gfCNCPoint1[14456] = {X 450.4384, Y 41.0287, Z -1.3333, A 0.000, B 0.000, C 0.000 }
gfCNCPoint1[14457] = {X 450.4384, Y 34.2338, Z -1.3333, A 0.000, B 0.000, C 0.000 }
gfCNCPoint1[14458] = {X 447.3268, Y 34.2338, Z -1.3333, A 0.000, B 0.000, C 0.000 }
gfCNCPoint1[14459] = {X 442.9270, Y 42.8001, Z -1.3333, A 0.000, B 0.000, C 0.000 }
gfCNCPoint1[14460] = {X 442.9680, Y 42.9095, Z -1.3333, A 0.000, B 0.000, C 0.000 }
gfCNCPoint1[14461] = {X 443.1240, Y 43.5326, Z -1.3333, A 0.000, B 0.000, C 0.000 }
gfCNCPoint1[14462] = {X 443.1803, Y 44.1725, Z -1.3333, A 0.000, B 0.000, C 0.000 }
gfCNCPoint1[14463] = {X 443.1805, Y 45.0000, Z -1.3333, A 0.000, B 0.000, C 0.000 }
gfCNCPoint1[14464] = {X 443.0782, Y 45.9079, Z -1.3333, A 0.000, B 0.000, C 0.000 }
gfCNCPoint1[14465] = {X 442.7764, Y 46.7702, Z -1.3333, A 0.000, B 0.000, C 0.000 }
gfCNCPoint1[14466] = {X 442.2903, Y 47.5438, Z -1.3333, A 0.000, B 0.000, C 0.000 }
gfCNCPoint1[14467] = {X 441.6443, Y 48.1899, Z -1.3333, A 0.000, B 0.000, C 0.000 }
gfCNCPoint1[14468] = {X 440.8707, Y 48.6760, Z -1.3333, A 0.000, B 0.000, C 0.000 }
gfCNCPoint1[14469] = {X 440.0084, Y 48.9777, Z -1.3333, A 0.000, B 0.000, C 0.000 }
gfCNCPoint1[14470] = {X 439.1005, Y 49.0800, Z -1.3333, A 0.000, B 0.000, C 0.000 }
gfCNCPoint1[14471] = {X 432.5144, Y 49.0800, Z -1.3333, A 0.000, B 0.000, C 0.000 }
gfCNCPoint1[14472] = {X 431.6065, Y 48.9777, Z -1.3333, A 0.000, B 0.000, C 0.000 }
gfCNCPoint1[14473] = {X 430.7442, Y 48.6760, Z -1.3333, A 0.000, B 0.000, C 0.000 }
gfCNCPoint1[14474] = {X 429.9706, Y 48.1899, Z -1.3333, A 0.000, B 0.000, C 0.000 }
gfCNCPoint1[14475] = {X 429.3245, Y 47.5438, Z -1.3333, A 0.000, B 0.000, C 0.000 }
gfCNCPoint1[14476] = {X 428.8385, Y 46.7702, Z -1.3333, A 0.000, B 0.000, C 0.000 }
gfCNCPoint1[14477] = {X 428.5367, Y 45.9079, Z -1.3333, A 0.000, B 0.000, C 0.000 }
gfCNCPoint1[14478] = {X 428.4344, Y 45.0000, Z -1.3333, A 0.000, B 0.000, C 0.000 }
gfCNCPoint1[14479] = {X 428.4348, Y 44.1527, Z -1.3333, A 0.000, B 0.000, C 0.000 }
gfCNCPoint1[14480] = {X 428.5303, Y 43.3294, Z -1.3333, A 0.000, B 0.000, C 0.000 }
gfCNCPoint1[14481] = {X 428.7902, Y 42.5424, Z -1.3333, A 0.000, B 0.000, C 0.000 }
gfCNCPoint1[14482] = {X 429.2038, Y 41.8242, Z -1.3333, A 0.000, B 0.000, C 0.000 }
gfCNCPoint1[14483] = {X 429.7540, Y 41.2044, Z -1.3333, A 0.000, B 0.000, C 0.000 }
gfCNCPoint1[14484] = {X 430.4181, Y 40.7085, Z -1.3333, A 0.000, B 0.000, C 0.000 }
gfCNCPoint1[14485] = {X 431.1687, Y 40.3571, Z -1.3333, A 0.000, B 0.000, C 0.000 }
gfCNCPoint1[14486] = {X 435.3054, Y 32.2601, Z -1.3333, A 0.000, B 0.000, C 0.000 }
gfCNCPoint1[14487] = {X 434.1145, Y 31.4915, Z -1.3333, A 0.000, B 0.000, C 0.000 }
gfCNCPoint1[14488] = {X 433.0315, Y 30.5771, Z -1.3333, A 0.000, B 0.000, C 0.000 }
gfCNCPoint1[14489] = {X 432.0741, Y 29.5320, Z -1.3333, A 0.000, B 0.000, C 0.000 }
gfCNCPoint1[14490] = {X 431.2580, Y 28.3732, Z -1.3333, A 0.000, B 0.000, C 0.000 }
gfCNCPoint1[14491] = {X 430.5964, Y 27.1197, Z -1.3333, A 0.000, B 0.000, C 0.000 }
gfCNCPoint1[14492] = {X 430.1003, Y 25.7920, Z -1.3333, A 0.000, B 0.000, C 0.000 }
gfCNCPoint1[14493] = {X 429.6876, Y 24.0071, Z -1.3333, A 0.000, B 0.000, C 0.000 }
gfCNCPoint1[14494] = {X 429.4774, Y 22.1872, Z -1.3333, A 0.000, B 0.000, C 0.000 }
gfCNCPoint1[14495] = {X 429.4722, Y 20.3552, Z -1.3333, A 0.000, B 0.000, C 0.000 }
gfCNCPoint1[14496] = {X 429.6722, Y 18.5341, Z -1.3333, A 0.000, B 0.000, C 0.000 }
gfCNCPoint1[14497] = {X 430.0749, Y 16.7469, Z -1.3333, A 0.000, B 0.000, C 0.000 }
gfCNCPoint1[14498] = {X 430.5856, Y 15.3070, Z -1.3333, A 0.000, B 0.000, C 0.000 }
gfCNCPoint1[14499] = {X 431.2819, Y 13.9471, Z -1.3333, A 0.000, B 0.000, C 0.000 }
gfCNCPoint1[14500] = {X 432.1516, Y 12.6910, Z -1.3333, A 0.000, B 0.000, C 0.000 }
gfCNCPoint1[14501] = {X 433.1794, Y 11.5607, Z -1.3333, A 0.000, B 0.000, C 0.000 }
gfCNCPoint1[14502] = {X 434.3473, Y 10.5759, Z -1.3333, A 0.000, B 0.000, C 0.000 }
gfCNCPoint1[14503] = {X 435.6351, Y 9.7538, Z -1.3333, A 0.000, B 0.000, C 0.000 }
gfCNCPoint1[14504] = {X 437.0200, Y 9.1088, Z -1.3333, A 0.000, B 0.000, C 0.000 }
gfCNCPoint1[14505] = {X 438.4780, Y 8.6523, Z -1.3333, A 0.000, B 0.000, C 0.000 }
gfCNCPoint1[14506] = {X 440.0844, Y 8.3468, Z -1.3333, A 0.000, B 0.000, C 0.000 }
gfCNCPoint1[14507] = {X 441.7098, Y 8.1677, Z -1.3333, A 0.000, B 0.000, C 0.000 }
gfCNCPoint1[14508] = {X 443.3442, Y 8.1160, Z -1.3333, A 0.000, B 0.000, C 0.000 }
gfCNCPoint1[14509] = {X 444.0364, Y 8.1119, Z -1.3333, A 0.000, B 0.000, C 0.000 }
gfCNCPoint1[14510] = {X 459.4465, Y 8.1119, Z -1.3333, A 0.000, B 0.000, C 0.000 }
gfCNCPoint1[14511] = {X 460.3525, Y 8.2140, Z -1.3333, A 0.000, B 0.000, C 0.000 }
gfCNCPoint1[14512] = {X 461.2130, Y 8.5151, Z -1.3333, A 0.000, B 0.000, C 0.000 }
gfCNCPoint1[14513] = {X 461.9850, Y 9.0002, Z -1.3333, A 0.000, B 0.000, C 0.000 }
gfCNCPoint1[14514] = {X 462.6297, Y 9.6448, Z -1.3333, A 0.000, B 0.000, C 0.000 }
gfCNCPoint1[14515] = {X 463.1147, Y 10.4168, Z -1.3333, A 0.000, B 0.000, C 0.000 }
gfCNCPoint1[14516] = {X 463.4159, Y 11.2774, Z -1.3333, A 0.000, B 0.000, C 0.000 }
gfCNCPoint1[14517] = {X 463.5179, Y 12.1834, Z -1.3333, A 0.000, B 0.000, C 0.000 }
gfCNCPoint1[14518] = {X 463.5179, Y 12.9781, Z -1.3333, A 0.000, B 0.000, C 0.000 }
gfCNCPoint1[14519] = {X 463.4240, Y 13.8483, Z -1.3333, A 0.000, B 0.000, C 0.000 }
gfCNCPoint1[14520] = {X 463.1467, Y 14.6785, Z -1.3333, A 0.000, B 0.000, C 0.000 }
gfCNCPoint1[14521] = {X 462.6987, Y 15.4304, Z -1.3333, A 0.000, B 0.000, C 0.000 }
gfCNCPoint1[14522] = {X 462.1006, Y 16.0694, Z -1.3333, A 0.000, B 0.000, C 0.000 }
gfCNCPoint1[14523] = {X 462.0432, Y 16.1179, Z -1.3333, A 0.000, B 0.000, C 0.000 }
gfCNCPoint1[14524] = {X 461.9850, Y 16.1653, Z -1.3333, A 0.000, B 0.000, C 0.000 }
gfCNCPoint1[14525] = {X 461.9894, Y 16.2000, Z -1.3333, A 0.000, B 0.000, C 0.000 }
gfCNCPoint1[14526] = {X 461.9896, Y 28.5936, Z -1.3333, A 0.000, B 0.000, C 0.000 }
gfCNCPoint1[14527] = {X 465.9896, Y 28.5935, Z -1.3333, A 0.000, B 0.000, C 0.000 }
gfCNCPoint1[14528] = {X 461.9096, Y 28.5936, Z -1.3333, A 0.000, B 0.000, C 0.000 }
gfCNCPoint1[14529] = {X 461.9098, Y 41.0659, Z -1.3333, A 0.000, B 0.000, C 0.000 }
gfCNCPoint1[14530] = {X 462.0488, Y 41.1783, Z -1.3333, A 0.000, B 0.000, C 0.000 }
gfCNCPoint1[14531] = {X 462.6350, Y 41.8049, Z -1.3333, A 0.000, B 0.000, C 0.000 }
gfCNCPoint1[14532] = {X 463.0741, Y 42.5420, Z -1.3333, A 0.000, B 0.000, C 0.000 }
gfCNCPoint1[14533] = {X 463.3459, Y 43.3558, Z -1.3333, A 0.000, B 0.000, C 0.000 }
gfCNCPoint1[14534] = {X 463.4379, Y 44.2089, Z -1.3333, A 0.000, B 0.000, C 0.000 }
gfCNCPoint1[14535] = {X 463.4379, Y 45.0000, Z -1.3333, A 0.000, B 0.000, C 0.000 }
gfCNCPoint1[14536] = {X 463.3377, Y 45.8901, Z -1.3333, A 0.000, B 0.000, C 0.000 }
gfCNCPoint1[14537] = {X 463.0418, Y 46.7355, Z -1.3333, A 0.000, B 0.000, C 0.000 }
gfCNCPoint1[14538] = {X 462.5653, Y 47.4940, Z -1.3333, A 0.000, B 0.000, C 0.000 }
gfCNCPoint1[14539] = {X 461.9319, Y 48.1273, Z -1.3333, A 0.000, B 0.000, C 0.000 }
gfCNCPoint1[14540] = {X 461.1735, Y 48.6039, Z -1.3333, A 0.000, B 0.000, C 0.000 }
gfCNCPoint1[14541] = {X 460.3280, Y 48.8997, Z -1.3333, A 0.000, B 0.000, C 0.000 }
gfCNCPoint1[14542] = {X 459.4379, Y 49.0000, Z -1.3333, A 0.000, B 0.000, C 0.000 }
gfCNCPoint1[14543] = {X 452.9945, Y 49.0000, Z -1.3333, A 0.000, B 0.000, C 0.000 }
gfCNCPoint1[14544] = {X 452.1044, Y 48.8997, Z -1.3333, A 0.000, B 0.000, C 0.000 }
gfCNCPoint1[14545] = {X 451.2589, Y 48.6039, Z -1.3333, A 0.000, B 0.000, C 0.000 }
gfCNCPoint1[14546] = {X 450.5005, Y 48.1273, Z -1.3333, A 0.000, B 0.000, C 0.000 }
gfCNCPoint1[14547] = {X 449.8671, Y 47.4939, Z -1.3333, A 0.000, B 0.000, C 0.000 }
gfCNCPoint1[14548] = {X 449.3906, Y 46.7355, Z -1.3333, A 0.000, B 0.000, C 0.000 }
gfCNCPoint1[14549] = {X 449.0948, Y 45.8900, Z -1.3333, A 0.000, B 0.000, C 0.000 }
gfCNCPoint1[14550] = {X 448.9945, Y 44.9999, Z -1.3333, A 0.000, B 0.000, C 0.000 }
gfCNCPoint1[14551] = {X 448.9949, Y 44.1538, Z -1.3333, A 0.000, B 0.000, C 0.000 }
gfCNCPoint1[14552] = {X 449.1055, Y 43.2730, Z -1.3333, A 0.000, B 0.000, C 0.000 }
gfCNCPoint1[14553] = {X 449.4077, Y 42.4382, Z -1.3333, A 0.000, B 0.000, C 0.000 }
gfCNCPoint1[14554] = {X 449.8865, Y 41.6907, Z -1.3333, A 0.000, B 0.000, C 0.000 }
gfCNCPoint1[14555] = {X 450.5184, Y 41.0672, Z -1.3333, A 0.000, B 0.000, C 0.000 }
gfCNCPoint1[14556] = {X 450.5184, Y 34.1538, Z -1.3333, A 0.000, B 0.000, C 0.000 }
gfCNCPoint1[14557] = {X 447.5222, Y 34.1538, Z -1.3333, A 0.000, B 0.000, C 0.000 }
gfCNCPoint1[14558] = {X 447.2789, Y 34.1521, Z -1.3333, A 0.000, B 0.000, C 0.000 }
gfCNCPoint1[14559] = {X 442.8397, Y 42.7950, Z -1.3333, A 0.000, B 0.000, C 0.000 }
gfCNCPoint1[14560] = {X 442.8963, Y 42.9473, Z -1.3333, A 0.000, B 0.000, C 0.000 }
gfCNCPoint1[14561] = {X 443.0491, Y 43.5699, Z -1.3333, A 0.000, B 0.000, C 0.000 }
gfCNCPoint1[14562] = {X 443.1005, Y 44.2089, Z -1.3333, A 0.000, B 0.000, C 0.000 }
gfCNCPoint1[14563] = {X 443.1005, Y 45.0000, Z -1.3333, A 0.000, B 0.000, C 0.000 }
gfCNCPoint1[14564] = {X 443.0002, Y 45.8901, Z -1.3333, A 0.000, B 0.000, C 0.000 }
gfCNCPoint1[14565] = {X 442.7043, Y 46.7355, Z -1.3333, A 0.000, B 0.000, C 0.000 }
gfCNCPoint1[14566] = {X 442.2278, Y 47.4940, Z -1.3333, A 0.000, B 0.000, C 0.000 }
gfCNCPoint1[14567] = {X 441.5944, Y 48.1273, Z -1.3333, A 0.000, B 0.000, C 0.000 }
gfCNCPoint1[14568] = {X 440.8360, Y 48.6039, Z -1.3333, A 0.000, B 0.000, C 0.000 }
gfCNCPoint1[14569] = {X 439.9906, Y 48.8997, Z -1.3333, A 0.000, B 0.000, C 0.000 }
gfCNCPoint1[14570] = {X 439.1005, Y 49.0000, Z -1.3333, A 0.000, B 0.000, C 0.000 }
gfCNCPoint1[14571] = {X 432.5144, Y 49.0000, Z -1.3333, A 0.000, B 0.000, C 0.000 }
gfCNCPoint1[14572] = {X 431.6243, Y 48.8997, Z -1.3333, A 0.000, B 0.000, C 0.000 }
gfCNCPoint1[14573] = {X 430.7789, Y 48.6039, Z -1.3333, A 0.000, B 0.000, C 0.000 }
gfCNCPoint1[14574] = {X 430.0204, Y 48.1273, Z -1.3333, A 0.000, B 0.000, C 0.000 }
gfCNCPoint1[14575] = {X 429.3871, Y 47.4940, Z -1.3333, A 0.000, B 0.000, C 0.000 }
gfCNCPoint1[14576] = {X 428.9105, Y 46.7355, Z -1.3333, A 0.000, B 0.000, C 0.000 }
gfCNCPoint1[14577] = {X 428.6147, Y 45.8901, Z -1.3333, A 0.000, B 0.000, C 0.000 }
gfCNCPoint1[14578] = {X 428.5144, Y 45.0000, Z -1.3333, A 0.000, B 0.000, C 0.000 }
gfCNCPoint1[14579] = {X 428.5148, Y 44.1538, Z -1.3333, A 0.000, B 0.000, C 0.000 }
gfCNCPoint1[14580] = {X 428.6096, Y 43.3414, Z -1.3333, A 0.000, B 0.000, C 0.000 }
gfCNCPoint1[14581] = {X 428.8676, Y 42.5654, Z -1.3333, A 0.000, B 0.000, C 0.000 }
gfCNCPoint1[14582] = {X 429.2781, Y 41.8580, Z -1.3333, A 0.000, B 0.000, C 0.000 }
gfCNCPoint1[14583] = {X 429.8239, Y 41.2489, Z -1.3333, A 0.000, B 0.000, C 0.000 }
gfCNCPoint1[14584] = {X 430.4821, Y 40.7635, Z -1.3333, A 0.000, B 0.000, C 0.000 }
gfCNCPoint1[14585] = {X 431.2253, Y 40.4222, Z -1.3333, A 0.000, B 0.000, C 0.000 }
gfCNCPoint1[14586] = {X 435.4118, Y 32.2276, Z -1.3333, A 0.000, B 0.000, C 0.000 }
gfCNCPoint1[14587] = {X 434.2139, Y 31.4652, Z -1.3333, A 0.000, B 0.000, C 0.000 }
gfCNCPoint1[14588] = {X 433.1241, Y 30.5549, Z -1.3333, A 0.000, B 0.000, C 0.000 }
gfCNCPoint1[14589] = {X 432.1607, Y 29.5118, Z -1.3333, A 0.000, B 0.000, C 0.000 }
gfCNCPoint1[14590] = {X 431.3397, Y 28.3533, Z -1.3333, A 0.000, B 0.000, C 0.000 }
gfCNCPoint1[14591] = {X 430.6747, Y 27.0987, Z -1.3333, A 0.000, B 0.000, C 0.000 }
gfCNCPoint1[14592] = {X 430.1769, Y 25.7689, Z -1.3333, A 0.000, B 0.000, C 0.000 }
gfCNCPoint1[14593] = {X 429.7663, Y 23.9928, Z -1.3333, A 0.000, B 0.000, C 0.000 }
gfCNCPoint1[14594] = {X 429.5572, Y 22.1819, Z -1.3333, A 0.000, B 0.000, C 0.000 }
gfCNCPoint1[14595] = {X 429.5521, Y 20.3591, Z -1.3333, A 0.000, B 0.000, C 0.000 }
gfCNCPoint1[14596] = {X 429.7512, Y 18.5471, Z -1.3333, A 0.000, B 0.000, C 0.000 }
gfCNCPoint1[14597] = {X 430.1519, Y 16.7687, Z -1.3333, A 0.000, B 0.000, C 0.000 }
gfCNCPoint1[14598] = {X 430.6590, Y 15.3388, Z -1.3333, A 0.000, B 0.000, C 0.000 }
gfCNCPoint1[14599] = {X 431.3505, Y 13.9883, Z -1.3333, A 0.000, B 0.000, C 0.000 }
gfCNCPoint1[14600] = {X 432.2141, Y 12.7409, Z -1.3333, A 0.000, B 0.000, C 0.000 }
gfCNCPoint1[14601] = {X 433.2348, Y 11.6184, Z -1.3333, A 0.000, B 0.000, C 0.000 }
gfCNCPoint1[14602] = {X 434.3947, Y 10.6403, Z -1.3333, A 0.000, B 0.000, C 0.000 }
gfCNCPoint1[14603] = {X 435.6735, Y 9.8239, Z -1.3333, A 0.000, B 0.000, C 0.000 }
gfCNCPoint1[14604] = {X 437.0489, Y 9.1834, Z -1.3333, A 0.000, B 0.000, C 0.000 }
gfCNCPoint1[14605] = {X 438.4968, Y 8.7301, Z -1.3333, A 0.000, B 0.000, C 0.000 }
gfCNCPoint1[14606] = {X 440.0970, Y 8.4258, Z -1.3333, A 0.000, B 0.000, C 0.000 }
gfCNCPoint1[14607] = {X 441.7161, Y 8.2474, Z -1.3333, A 0.000, B 0.000, C 0.000 }
gfCNCPoint1[14608] = {X 443.3442, Y 8.1960, Z -1.3333, A 0.000, B 0.000, C 0.000 }
gfCNCPoint1[14609] = {X 444.0367, Y 8.1919, Z -1.3333, A 0.000, B 0.000, C 0.000 }
gfCNCPoint1[14610] = {X 459.4465, Y 8.1919, Z -1.3333, A 0.000, B 0.000, C 0.000 }
gfCNCPoint1[14611] = {X 460.3347, Y 8.2920, Z -1.3333, A 0.000, B 0.000, C 0.000 }
gfCNCPoint1[14612] = {X 461.1783, Y 8.5872, Z -1.3333, A 0.000, B 0.000, C 0.000 }
gfCNCPoint1[14613] = {X 461.9351, Y 9.0627, Z -1.3333, A 0.000, B 0.000, C 0.000 }
gfCNCPoint1[14614] = {X 462.5671, Y 9.6947, Z -1.3333, A 0.000, B 0.000, C 0.000 }
gfCNCPoint1[14615] = {X 463.0427, Y 10.4515, Z -1.3333, A 0.000, B 0.000, C 0.000 }
gfCNCPoint1[14616] = {X 463.3379, Y 11.2952, Z -1.3333, A 0.000, B 0.000, C 0.000 }
gfCNCPoint1[14617] = {X 463.4379, Y 12.1834, Z -1.3333, A 0.000, B 0.000, C 0.000 }
gfCNCPoint1[14618] = {X 463.4378, Y 13.0163, Z -1.3333, A 0.000, B 0.000, C 0.000 }
gfCNCPoint1[14619] = {X 463.3397, Y 13.8592, Z -1.3333, A 0.000, B 0.000, C 0.000 }
gfCNCPoint1[14620] = {X 463.0660, Y 14.6625, Z -1.3333, A 0.000, B 0.000, C 0.000 }
gfCNCPoint1[14621] = {X 462.6290, Y 15.3899, Z -1.3333, A 0.000, B 0.000, C 0.000 }
gfCNCPoint1[14622] = {X 462.0484, Y 16.0088, Z -1.3333, A 0.000, B 0.000, C 0.000 }
gfCNCPoint1[14623] = {X 461.9721, Y 16.0729, Z -1.3333, A 0.000, B 0.000, C 0.000 }
gfCNCPoint1[14624] = {X 461.8942, Y 16.1351, Z -1.3333, A 0.000, B 0.000, C 0.000 }
gfCNCPoint1[14625] = {X 461.9094, Y 16.1924, Z -1.3333, A 0.000, B 0.000, C 0.000 }
gfCNCPoint1[14626] = {X 461.9096, Y 28.5936, Z -1.3333, A 0.000, B 0.000, C 0.000 }
gfCNCPoint1[14627] = {X 465.9896, Y 28.5935, Z -1.3333, A 0.000, B 0.000, C 0.000 }
gfCNCPoint1[14628] = {X 465.9896, Y 28.5935, Z 1.6667, A 0.000, B 0.000, C 0.000 }
gfCNCPoint1[14629] = {X 465.9896, Y 28.5935, Z 11.0000, A 0.000, B 0.000, C 0.000 }
gfCNCPoint1[14630] = {X 492.3824, Y 3.7919, Z 11.0000, A 0.000, B 0.000, C 0.000 }
gfCNCPoint1[14631] = {X 492.3824, Y 3.7919, Z 1.6667, A 0.000, B 0.000, C 0.000 }
gfCNCPoint1[14632] = {X 492.3824, Y 3.7919, Z -1.3333, A 0.000, B 0.000, C 0.000 }
gfCNCPoint1[14633] = {X 492.3824, Y 7.8719, Z -1.3333, A 0.000, B 0.000, C 0.000 }
gfCNCPoint1[14634] = {X 502.2066, Y 7.8719, Z -1.3333, A 0.000, B 0.000, C 0.000 }
gfCNCPoint1[14635] = {X 502.7373, Y 7.8760, Z -1.3333, A 0.000, B 0.000, C 0.000 }
gfCNCPoint1[14636] = {X 503.6897, Y 7.9904, Z -1.3333, A 0.000, B 0.000, C 0.000 }
gfCNCPoint1[14637] = {X 504.5931, Y 8.3127, Z -1.3333, A 0.000, B 0.000, C 0.000 }
gfCNCPoint1[14638] = {X 505.4027, Y 8.8271, Z -1.3333, A 0.000, B 0.000, C 0.000 }
gfCNCPoint1[14639] = {X 506.0783, Y 9.5080, Z -1.3333, A 0.000, B 0.000, C 0.000 }
gfCNCPoint1[14640] = {X 506.5863, Y 10.3216, Z -1.3333, A 0.000, B 0.000, C 0.000 }
gfCNCPoint1[14641] = {X 506.9016, Y 11.2275, Z -1.3333, A 0.000, B 0.000, C 0.000 }
gfCNCPoint1[14642] = {X 507.0085, Y 12.1807, Z -1.3333, A 0.000, B 0.000, C 0.000 }
gfCNCPoint1[14643] = {X 507.0085, Y 12.9781, Z -1.3333, A 0.000, B 0.000, C 0.000 }
gfCNCPoint1[14644] = {X 506.9071, Y 13.9084, Z -1.3333, A 0.000, B 0.000, C 0.000 }
gfCNCPoint1[14645] = {X 506.6078, Y 14.7951, Z -1.3333, A 0.000, B 0.000, C 0.000 }
gfCNCPoint1[14646] = {X 506.1245, Y 15.5965, Z -1.3333, A 0.000, B 0.000, C 0.000 }
gfCNCPoint1[14647] = {X 505.4800, Y 16.2750, Z -1.3333, A 0.000, B 0.000, C 0.000 }
gfCNCPoint1[14648] = {X 505.4799, Y 40.9118, Z -1.3333, A 0.000, B 0.000, C 0.000 }
gfCNCPoint1[14649] = {X 506.1188, Y 41.5829, Z -1.3333, A 0.000, B 0.000, C 0.000 }
gfCNCPoint1[14650] = {X 506.5998, Y 42.3747, Z -1.3333, A 0.000, B 0.000, C 0.000 }
gfCNCPoint1[14651] = {X 506.9010, Y 43.2510, Z -1.3333, A 0.000, B 0.000, C 0.000 }
gfCNCPoint1[14652] = {X 507.0083, Y 44.1713, Z -1.3333, A 0.000, B 0.000, C 0.000 }
gfCNCPoint1[14653] = {X 507.0085, Y 45.0000, Z -1.3333, A 0.000, B 0.000, C 0.000 }
gfCNCPoint1[14654] = {X 506.9002, Y 45.9613, Z -1.3333, A 0.000, B 0.000, C 0.000 }
gfCNCPoint1[14655] = {X 506.5807, Y 46.8744, Z -1.3333, A 0.000, B 0.000, C 0.000 }
gfCNCPoint1[14656] = {X 506.0660, Y 47.6935, Z -1.3333, A 0.000, B 0.000, C 0.000 }
gfCNCPoint1[14657] = {X 505.3820, Y 48.3775, Z -1.3333, A 0.000, B 0.000, C 0.000 }
gfCNCPoint1[14658] = {X 504.5629, Y 48.8922, Z -1.3333, A 0.000, B 0.000, C 0.000 }
gfCNCPoint1[14659] = {X 503.6498, Y 49.2117, Z -1.3333, A 0.000, B 0.000, C 0.000 }
gfCNCPoint1[14660] = {X 502.6885, Y 49.3200, Z -1.3333, A 0.000, B 0.000, C 0.000 }
gfCNCPoint1[14661] = {X 496.2450, Y 49.3200, Z -1.3333, A 0.000, B 0.000, C 0.000 }
gfCNCPoint1[14662] = {X 495.2885, Y 49.2128, Z -1.3333, A 0.000, B 0.000, C 0.000 }
gfCNCPoint1[14663] = {X 494.3794, Y 48.8964, Z -1.3333, A 0.000, B 0.000, C 0.000 }
gfCNCPoint1[14664] = {X 493.5630, Y 48.3866, Z -1.3333, A 0.000, B 0.000, C 0.000 }
gfCNCPoint1[14665] = {X 492.8797, Y 47.7087, Z -1.3333, A 0.000, B 0.000, C 0.000 }
gfCNCPoint1[14666] = {X 492.3635, Y 46.8963, Z -1.3333, A 0.000, B 0.000, C 0.000 }
gfCNCPoint1[14667] = {X 492.0399, Y 45.9898, Z -1.3333, A 0.000, B 0.000, C 0.000 }
gfCNCPoint1[14668] = {X 491.9252, Y 45.0341, Z -1.3333, A 0.000, B 0.000, C 0.000 }
gfCNCPoint1[14669] = {X 491.9254, Y 44.1494, Z -1.3333, A 0.000, B 0.000, C 0.000 }
gfCNCPoint1[14670] = {X 492.0359, Y 43.2364, Z -1.3333, A 0.000, B 0.000, C 0.000 }
gfCNCPoint1[14671] = {X 492.3371, Y 42.3675, Z -1.3333, A 0.000, B 0.000, C 0.000 }
gfCNCPoint1[14672] = {X 492.8153, Y 41.5821, Z -1.3333, A 0.000, B 0.000, C 0.000 }
gfCNCPoint1[14673] = {X 493.4490, Y 40.9157, Z -1.3333, A 0.000, B 0.000, C 0.000 }
gfCNCPoint1[14674] = {X 493.4490, Y 34.4738, Z -1.3333, A 0.000, B 0.000, C 0.000 }
gfCNCPoint1[14675] = {X 490.7232, Y 34.4738, Z -1.3333, A 0.000, B 0.000, C 0.000 }
gfCNCPoint1[14676] = {X 486.4395, Y 42.8153, Z -1.3333, A 0.000, B 0.000, C 0.000 }
gfCNCPoint1[14677] = {X 486.4446, Y 42.8286, Z -1.3333, A 0.000, B 0.000, C 0.000 }
gfCNCPoint1[14678] = {X 486.6109, Y 43.4903, Z -1.3333, A 0.000, B 0.000, C 0.000 }
gfCNCPoint1[14679] = {X 486.6708, Y 44.1699, Z -1.3333, A 0.000, B 0.000, C 0.000 }
gfCNCPoint1[14680] = {X 486.6710, Y 45.0000, Z -1.3333, A 0.000, B 0.000, C 0.000 }
gfCNCPoint1[14681] = {X 486.5627, Y 45.9613, Z -1.3333, A 0.000, B 0.000, C 0.000 }
gfCNCPoint1[14682] = {X 486.2432, Y 46.8744, Z -1.3333, A 0.000, B 0.000, C 0.000 }
gfCNCPoint1[14683] = {X 485.7285, Y 47.6935, Z -1.3333, A 0.000, B 0.000, C 0.000 }
gfCNCPoint1[14684] = {X 485.0445, Y 48.3775, Z -1.3333, A 0.000, B 0.000, C 0.000 }
gfCNCPoint1[14685] = {X 484.2254, Y 48.8922, Z -1.3333, A 0.000, B 0.000, C 0.000 }
gfCNCPoint1[14686] = {X 483.3123, Y 49.2117, Z -1.3333, A 0.000, B 0.000, C 0.000 }
gfCNCPoint1[14687] = {X 482.3510, Y 49.3200, Z -1.3333, A 0.000, B 0.000, C 0.000 }
gfCNCPoint1[14688] = {X 475.7650, Y 49.3200, Z -1.3333, A 0.000, B 0.000, C 0.000 }
gfCNCPoint1[14689] = {X 474.8037, Y 49.2117, Z -1.3333, A 0.000, B 0.000, C 0.000 }
gfCNCPoint1[14690] = {X 473.8906, Y 48.8922, Z -1.3333, A 0.000, B 0.000, C 0.000 }
gfCNCPoint1[14691] = {X 473.0715, Y 48.3775, Z -1.3333, A 0.000, B 0.000, C 0.000 }
gfCNCPoint1[14692] = {X 472.3875, Y 47.6935, Z -1.3333, A 0.000, B 0.000, C 0.000 }
gfCNCPoint1[14693] = {X 471.8728, Y 46.8745, Z -1.3333, A 0.000, B 0.000, C 0.000 }
gfCNCPoint1[14694] = {X 471.5533, Y 45.9614, Z -1.3333, A 0.000, B 0.000, C 0.000 }
gfCNCPoint1[14695] = {X 471.4450, Y 45.0001, Z -1.3333, A 0.000, B 0.000, C 0.000 }
gfCNCPoint1[14696] = {X 471.4454, Y 44.1494, Z -1.3333, A 0.000, B 0.000, C 0.000 }
gfCNCPoint1[14697] = {X 471.5430, Y 43.2935, Z -1.3333, A 0.000, B 0.000, C 0.000 }
gfCNCPoint1[14698] = {X 471.8086, Y 42.4740, Z -1.3333, A 0.000, B 0.000, C 0.000 }
gfCNCPoint1[14699] = {X 472.2314, Y 41.7236, Z -1.3333, A 0.000, B 0.000, C 0.000 }
gfCNCPoint1[14700] = {X 472.7947, Y 41.0719, Z -1.3333, A 0.000, B 0.000, C 0.000 }
gfCNCPoint1[14701] = {X 473.4762, Y 40.5449, Z -1.3333, A 0.000, B 0.000, C 0.000 }
gfCNCPoint1[14702] = {X 474.2486, Y 40.1637, Z -1.3333, A 0.000, B 0.000, C 0.000 }
gfCNCPoint1[14703] = {X 478.2331, Y 32.3645, Z -1.3333, A 0.000, B 0.000, C 0.000 }
gfCNCPoint1[14704] = {X 476.9699, Y 31.4967, Z -1.3333, A 0.000, B 0.000, C 0.000 }
gfCNCPoint1[14705] = {X 475.8338, Y 30.4682, Z -1.3333, A 0.000, B 0.000, C 0.000 }
gfCNCPoint1[14706] = {X 474.8448, Y 29.2975, Z -1.3333, A 0.000, B 0.000, C 0.000 }
gfCNCPoint1[14707] = {X 474.0207, Y 28.0054, Z -1.3333, A 0.000, B 0.000, C 0.000 }
gfCNCPoint1[14708] = {X 473.3762, Y 26.6150, Z -1.3333, A 0.000, B 0.000, C 0.000 }
gfCNCPoint1[14709] = {X 472.9228, Y 25.1511, Z -1.3333, A 0.000, B 0.000, C 0.000 }
gfCNCPoint1[14710] = {X 472.6086, Y 23.4680, Z -1.3333, A 0.000, B 0.000, C 0.000 }
gfCNCPoint1[14711] = {X 472.4681, Y 21.7616, Z -1.3333, A 0.000, B 0.000, C 0.000 }
gfCNCPoint1[14712] = {X 472.5028, Y 20.0497, Z -1.3333, A 0.000, B 0.000, C 0.000 }
gfCNCPoint1[14713] = {X 472.7123, Y 18.3504, Z -1.3333, A 0.000, B 0.000, C 0.000 }
gfCNCPoint1[14714] = {X 473.0945, Y 16.6814, Z -1.3333, A 0.000, B 0.000, C 0.000 }
gfCNCPoint1[14715] = {X 473.6376, Y 15.1671, Z -1.3333, A 0.000, B 0.000, C 0.000 }
gfCNCPoint1[14716] = {X 474.3811, Y 13.7404, Z -1.3333, A 0.000, B 0.000, C 0.000 }
gfCNCPoint1[14717] = {X 475.3112, Y 12.4277, Z -1.3333, A 0.000, B 0.000, C 0.000 }
gfCNCPoint1[14718] = {X 476.4106, Y 11.2533, Z -1.3333, A 0.000, B 0.000, C 0.000 }
gfCNCPoint1[14719] = {X 477.6592, Y 10.2388, Z -1.3333, A 0.000, B 0.000, C 0.000 }
gfCNCPoint1[14720] = {X 479.0338, Y 9.4030, Z -1.3333, A 0.000, B 0.000, C 0.000 }
gfCNCPoint1[14721] = {X 480.5091, Y 8.7613, Z -1.3333, A 0.000, B 0.000, C 0.000 }
gfCNCPoint1[14722] = {X 482.0578, Y 8.3256, Z -1.3333, A 0.000, B 0.000, C 0.000 }
gfCNCPoint1[14723] = {X 484.1551, Y 7.9992, Z -1.3333, A 0.000, B 0.000, C 0.000 }
gfCNCPoint1[14724] = {X 486.2746, Y 7.8841, Z -1.3333, A 0.000, B 0.000, C 0.000 }
gfCNCPoint1[14725] = {X 486.9679, Y 7.8719, Z -1.3333, A 0.000, B 0.000, C 0.000 }
gfCNCPoint1[14726] = {X 492.3824, Y 7.8719, Z -1.3333, A 0.000, B 0.000, C 0.000 }
gfCNCPoint1[14727] = {X 492.3824, Y 3.8719, Z -1.3333, A 0.000, B 0.000, C 0.000 }
gfCNCPoint1[14728] = {X 492.3824, Y 7.9519, Z -1.3333, A 0.000, B 0.000, C 0.000 }
gfCNCPoint1[14729] = {X 502.2063, Y 7.9519, Z -1.3333, A 0.000, B 0.000, C 0.000 }
gfCNCPoint1[14730] = {X 502.7367, Y 7.9560, Z -1.3333, A 0.000, B 0.000, C 0.000 }
gfCNCPoint1[14731] = {X 503.6713, Y 8.0682, Z -1.3333, A 0.000, B 0.000, C 0.000 }
gfCNCPoint1[14732] = {X 504.5580, Y 8.3846, Z -1.3333, A 0.000, B 0.000, C 0.000 }
gfCNCPoint1[14733] = {X 505.3525, Y 8.8894, Z -1.3333, A 0.000, B 0.000, C 0.000 }
gfCNCPoint1[14734] = {X 506.0156, Y 9.5577, Z -1.3333, A 0.000, B 0.000, C 0.000 }
gfCNCPoint1[14735] = {X 506.5142, Y 10.3562, Z -1.3333, A 0.000, B 0.000, C 0.000 }
gfCNCPoint1[14736] = {X 506.8236, Y 11.2452, Z -1.3333, A 0.000, B 0.000, C 0.000 }
gfCNCPoint1[14737] = {X 506.9285, Y 12.1807, Z -1.3333, A 0.000, B 0.000, C 0.000 }
gfCNCPoint1[14738] = {X 506.9285, Y 12.9781, Z -1.3333, A 0.000, B 0.000, C 0.000 }
gfCNCPoint1[14739] = {X 506.8270, Y 13.9002, Z -1.3333, A 0.000, B 0.000, C 0.000 }
gfCNCPoint1[14740] = {X 506.5274, Y 14.7782, Z -1.3333, A 0.000, B 0.000, C 0.000 }
gfCNCPoint1[14741] = {X 506.0440, Y 15.5700, Z -1.3333, A 0.000, B 0.000, C 0.000 }
gfCNCPoint1[14742] = {X 505.4000, Y 16.2377, Z -1.3333, A 0.000, B 0.000, C 0.000 }
gfCNCPoint1[14743] = {X 505.3999, Y 40.9499, Z -1.3333, A 0.000, B 0.000, C 0.000 }
gfCNCPoint1[14744] = {X 505.4282, Y 40.9728, Z -1.3333, A 0.000, B 0.000, C 0.000 }
gfCNCPoint1[14745] = {X 506.0553, Y 41.6315, Z -1.3333, A 0.000, B 0.000, C 0.000 }
gfCNCPoint1[14746] = {X 506.5274, Y 42.4087, Z -1.3333, A 0.000, B 0.000, C 0.000 }
gfCNCPoint1[14747] = {X 506.8230, Y 43.2687, Z -1.3333, A 0.000, B 0.000, C 0.000 }
gfCNCPoint1[14748] = {X 506.9283, Y 44.1720, Z -1.3333, A 0.000, B 0.000, C 0.000 }
gfCNCPoint1[14749] = {X 506.9285, Y 45.0000, Z -1.3333, A 0.000, B 0.000, C 0.000 }
gfCNCPoint1[14750] = {X 506.8222, Y 45.9435, Z -1.3333, A 0.000, B 0.000, C 0.000 }
gfCNCPoint1[14751] = {X 506.5086, Y 46.8397, Z -1.3333, A 0.000, B 0.000, C 0.000 }
gfCNCPoint1[14752] = {X 506.0035, Y 47.6436, Z -1.3333, A 0.000, B 0.000, C 0.000 }
gfCNCPoint1[14753] = {X 505.3321, Y 48.3150, Z -1.3333, A 0.000, B 0.000, C 0.000 }
gfCNCPoint1[14754] = {X 504.5282, Y 48.8201, Z -1.3333, A 0.000, B 0.000, C 0.000 }
gfCNCPoint1[14755] = {X 503.6320, Y 49.1337, Z -1.3333, A 0.000, B 0.000, C 0.000 }
gfCNCPoint1[14756] = {X 502.6885, Y 49.2400, Z -1.3333, A 0.000, B 0.000, C 0.000 }
gfCNCPoint1[14757] = {X 496.2450, Y 49.2400, Z -1.3333, A 0.000, B 0.000, C 0.000 }
gfCNCPoint1[14758] = {X 495.3062, Y 49.1348, Z -1.3333, A 0.000, B 0.000, C 0.000 }
gfCNCPoint1[14759] = {X 494.4140, Y 48.8242, Z -1.3333, A 0.000, B 0.000, C 0.000 }
gfCNCPoint1[14760] = {X 493.6127, Y 48.3239, Z -1.3333, A 0.000, B 0.000, C 0.000 }
gfCNCPoint1[14761] = {X 492.9420, Y 47.6585, Z -1.3333, A 0.000, B 0.000, C 0.000 }
gfCNCPoint1[14762] = {X 492.4354, Y 46.8612, Z -1.3333, A 0.000, B 0.000, C 0.000 }
gfCNCPoint1[14763] = {X 492.1178, Y 45.9714, Z -1.3333, A 0.000, B 0.000, C 0.000 }
gfCNCPoint1[14764] = {X 492.0052, Y 45.0335, Z -1.3333, A 0.000, B 0.000, C 0.000 }
gfCNCPoint1[14765] = {X 492.0054, Y 44.1505, Z -1.3333, A 0.000, B 0.000, C 0.000 }
gfCNCPoint1[14766] = {X 492.1159, Y 43.2454, Z -1.3333, A 0.000, B 0.000, C 0.000 }
gfCNCPoint1[14767] = {X 492.4173, Y 42.3850, Z -1.3333, A 0.000, B 0.000, C 0.000 }
gfCNCPoint1[14768] = {X 492.8957, Y 41.6088, Z -1.3333, A 0.000, B 0.000, C 0.000 }
gfCNCPoint1[14769] = {X 493.5290, Y 40.9529, Z -1.3333, A 0.000, B 0.000, C 0.000 }
gfCNCPoint1[14770] = {X 493.5290, Y 34.3938, Z -1.3333, A 0.000, B 0.000, C 0.000 }
gfCNCPoint1[14771] = {X 490.6743, Y 34.3938, Z -1.3333, A 0.000, B 0.000, C 0.000 }
gfCNCPoint1[14772] = {X 486.3520, Y 42.8106, Z -1.3333, A 0.000, B 0.000, C 0.000 }
gfCNCPoint1[14773] = {X 486.3693, Y 42.8558, Z -1.3333, A 0.000, B 0.000, C 0.000 }
gfCNCPoint1[14774] = {X 486.5321, Y 43.5044, Z -1.3333, A 0.000, B 0.000, C 0.000 }
gfCNCPoint1[14775] = {X 486.5908, Y 44.1706, Z -1.3333, A 0.000, B 0.000, C 0.000 }
gfCNCPoint1[14776] = {X 486.5910, Y 45.0000, Z -1.3333, A 0.000, B 0.000, C 0.000 }
gfCNCPoint1[14777] = {X 486.4847, Y 45.9435, Z -1.3333, A 0.000, B 0.000, C 0.000 }
gfCNCPoint1[14778] = {X 486.1711, Y 46.8397, Z -1.3333, A 0.000, B 0.000, C 0.000 }
gfCNCPoint1[14779] = {X 485.6660, Y 47.6436, Z -1.3333, A 0.000, B 0.000, C 0.000 }
gfCNCPoint1[14780] = {X 484.9946, Y 48.3150, Z -1.3333, A 0.000, B 0.000, C 0.000 }
gfCNCPoint1[14781] = {X 484.1907, Y 48.8201, Z -1.3333, A 0.000, B 0.000, C 0.000 }
gfCNCPoint1[14782] = {X 483.2945, Y 49.1337, Z -1.3333, A 0.000, B 0.000, C 0.000 }
gfCNCPoint1[14783] = {X 482.3510, Y 49.2400, Z -1.3333, A 0.000, B 0.000, C 0.000 }
gfCNCPoint1[14784] = {X 475.7650, Y 49.2400, Z -1.3333, A 0.000, B 0.000, C 0.000 }
gfCNCPoint1[14785] = {X 474.8215, Y 49.1337, Z -1.3333, A 0.000, B 0.000, C 0.000 }
gfCNCPoint1[14786] = {X 473.9253, Y 48.8201, Z -1.3333, A 0.000, B 0.000, C 0.000 }
gfCNCPoint1[14787] = {X 473.1214, Y 48.3150, Z -1.3333, A 0.000, B 0.000, C 0.000 }
gfCNCPoint1[14788] = {X 472.4500, Y 47.6436, Z -1.3333, A 0.000, B 0.000, C 0.000 }
gfCNCPoint1[14789] = {X 471.9449, Y 46.8397, Z -1.3333, A 0.000, B 0.000, C 0.000 }
gfCNCPoint1[14790] = {X 471.6313, Y 45.9436, Z -1.3333, A 0.000, B 0.000, C 0.000 }
gfCNCPoint1[14791] = {X 471.5250, Y 45.0001, Z -1.3333, A 0.000, B 0.000, C 0.000 }
gfCNCPoint1[14792] = {X 471.5254, Y 44.1505, Z -1.3333, A 0.000, B 0.000, C 0.000 }
gfCNCPoint1[14793] = {X 471.6223, Y 43.3054, Z -1.3333, A 0.000, B 0.000, C 0.000 }
gfCNCPoint1[14794] = {X 471.8860, Y 42.4967, Z -1.3333, A 0.000, B 0.000, C 0.000 }
gfCNCPoint1[14795] = {X 472.3057, Y 41.7570, Z -1.3333, A 0.000, B 0.000, C 0.000 }
gfCNCPoint1[14796] = {X 472.8647, Y 41.1159, Z -1.3333, A 0.000, B 0.000, C 0.000 }
gfCNCPoint1[14797] = {X 473.5404, Y 40.5992, Z -1.3333, A 0.000, B 0.000, C 0.000 }
gfCNCPoint1[14798] = {X 474.3057, Y 40.2278, Z -1.3333, A 0.000, B 0.000, C 0.000 }
gfCNCPoint1[14799] = {X 478.3386, Y 32.3337, Z -1.3333, A 0.000, B 0.000, C 0.000 }
gfCNCPoint1[14800] = {X 477.0688, Y 31.4726, Z -1.3333, A 0.000, B 0.000, C 0.000 }
gfCNCPoint1[14801] = {X 475.9261, Y 30.4485, Z -1.3333, A 0.000, B 0.000, C 0.000 }
gfCNCPoint1[14802] = {X 474.9315, Y 29.2802, Z -1.3333, A 0.000, B 0.000, C 0.000 }
gfCNCPoint1[14803] = {X 474.1029, Y 27.9889, Z -1.3333, A 0.000, B 0.000, C 0.000 }
gfCNCPoint1[14804] = {X 473.4553, Y 26.5979, Z -1.3333, A 0.000, B 0.000, C 0.000 }
gfCNCPoint1[14805] = {X 473.0006, Y 25.1325, Z -1.3333, A 0.000, B 0.000, C 0.000 }
gfCNCPoint1[14806] = {X 472.6879, Y 23.4574, Z -1.3333, A 0.000, B 0.000, C 0.000 }
gfCNCPoint1[14807] = {X 472.5481, Y 21.7591, Z -1.3333, A 0.000, B 0.000, C 0.000 }
gfCNCPoint1[14808] = {X 472.5826, Y 20.0555, Z -1.3333, A 0.000, B 0.000, C 0.000 }
gfCNCPoint1[14809] = {X 472.7911, Y 18.3643, Z -1.3333, A 0.000, B 0.000, C 0.000 }
gfCNCPoint1[14810] = {X 473.1715, Y 16.7033, Z -1.3333, A 0.000, B 0.000, C 0.000 }
gfCNCPoint1[14811] = {X 473.7109, Y 15.1992, Z -1.3333, A 0.000, B 0.000, C 0.000 }
gfCNCPoint1[14812] = {X 474.4494, Y 13.7821, Z -1.3333, A 0.000, B 0.000, C 0.000 }
gfCNCPoint1[14813] = {X 475.3731, Y 12.4783, Z -1.3333, A 0.000, B 0.000, C 0.000 }
gfCNCPoint1[14814] = {X 476.4652, Y 11.3118, Z -1.3333, A 0.000, B 0.000, C 0.000 }
gfCNCPoint1[14815] = {X 477.7053, Y 10.3042, Z -1.3333, A 0.000, B 0.000, C 0.000 }
gfCNCPoint1[14816] = {X 479.0707, Y 9.4740, Z -1.3333, A 0.000, B 0.000, C 0.000 }
gfCNCPoint1[14817] = {X 480.5360, Y 8.8366, Z -1.3333, A 0.000, B 0.000, C 0.000 }
gfCNCPoint1[14818] = {X 482.0741, Y 8.4039, Z -1.3333, A 0.000, B 0.000, C 0.000 }
gfCNCPoint1[14819] = {X 484.1638, Y 8.0787, Z -1.3333, A 0.000, B 0.000, C 0.000 }
gfCNCPoint1[14820] = {X 486.2755, Y 7.9641, Z -1.3333, A 0.000, B 0.000, C 0.000 }
gfCNCPoint1[14821] = {X 486.9686, Y 7.9519, Z -1.3333, A 0.000, B 0.000, C 0.000 }
gfCNCPoint1[14822] = {X 492.3824, Y 7.9519, Z -1.3333, A 0.000, B 0.000, C 0.000 }
gfCNCPoint1[14823] = {X 492.3824, Y 3.9519, Z -1.3333, A 0.000, B 0.000, C 0.000 }
gfCNCPoint1[14824] = {X 492.3824, Y 8.0319, Z -1.3333, A 0.000, B 0.000, C 0.000 }
gfCNCPoint1[14825] = {X 502.2059, Y 8.0319, Z -1.3333, A 0.000, B 0.000, C 0.000 }
gfCNCPoint1[14826] = {X 502.7360, Y 8.0360, Z -1.3333, A 0.000, B 0.000, C 0.000 }
gfCNCPoint1[14827] = {X 503.6530, Y 8.1461, Z -1.3333, A 0.000, B 0.000, C 0.000 }
gfCNCPoint1[14828] = {X 504.5228, Y 8.4565, Z -1.3333, A 0.000, B 0.000, C 0.000 }
gfCNCPoint1[14829] = {X 505.3024, Y 8.9518, Z -1.3333, A 0.000, B 0.000, C 0.000 }
gfCNCPoint1[14830] = {X 505.9529, Y 9.6073, Z -1.3333, A 0.000, B 0.000, C 0.000 }
gfCNCPoint1[14831] = {X 506.4420, Y 10.3907, Z -1.3333, A 0.000, B 0.000, C 0.000 }
gfCNCPoint1[14832] = {X 506.7456, Y 11.2629, Z -1.3333, A 0.000, B 0.000, C 0.000 }
gfCNCPoint1[14833] = {X 506.8485, Y 12.1807, Z -1.3333, A 0.000, B 0.000, C 0.000 }
gfCNCPoint1[14834] = {X 506.8485, Y 12.9781, Z -1.3333, A 0.000, B 0.000, C 0.000 }
gfCNCPoint1[14835] = {X 506.7469, Y 13.8919, Z -1.3333, A 0.000, B 0.000, C 0.000 }
gfCNCPoint1[14836] = {X 506.4470, Y 14.7611, Z -1.3333, A 0.000, B 0.000, C 0.000 }
gfCNCPoint1[14837] = {X 505.9635, Y 15.5432, Z -1.3333, A 0.000, B 0.000, C 0.000 }
gfCNCPoint1[14838] = {X 505.3200, Y 16.2000, Z -1.3333, A 0.000, B 0.000, C 0.000 }
gfCNCPoint1[14839] = {X 505.3199, Y 40.9886, Z -1.3333, A 0.000, B 0.000, C 0.000 }
gfCNCPoint1[14840] = {X 505.3673, Y 41.0261, Z -1.3333, A 0.000, B 0.000, C 0.000 }
gfCNCPoint1[14841] = {X 505.9862, Y 41.6730, Z -1.3333, A 0.000, B 0.000, C 0.000 }
gfCNCPoint1[14842] = {X 506.4524, Y 42.4372, Z -1.3333, A 0.000, B 0.000, C 0.000 }
gfCNCPoint1[14843] = {X 506.7443, Y 43.2835, Z -1.3333, A 0.000, B 0.000, C 0.000 }
gfCNCPoint1[14844] = {X 506.8483, Y 44.1727, Z -1.3333, A 0.000, B 0.000, C 0.000 }
gfCNCPoint1[14845] = {X 506.8485, Y 45.0000, Z -1.3333, A 0.000, B 0.000, C 0.000 }
gfCNCPoint1[14846] = {X 506.7442, Y 45.9257, Z -1.3333, A 0.000, B 0.000, C 0.000 }
gfCNCPoint1[14847] = {X 506.4365, Y 46.8050, Z -1.3333, A 0.000, B 0.000, C 0.000 }
gfCNCPoint1[14848] = {X 505.9409, Y 47.5937, Z -1.3333, A 0.000, B 0.000, C 0.000 }
gfCNCPoint1[14849] = {X 505.2822, Y 48.2524, Z -1.3333, A 0.000, B 0.000, C 0.000 }
gfCNCPoint1[14850] = {X 504.4934, Y 48.7480, Z -1.3333, A 0.000, B 0.000, C 0.000 }
gfCNCPoint1[14851] = {X 503.6142, Y 49.0557, Z -1.3333, A 0.000, B 0.000, C 0.000 }
gfCNCPoint1[14852] = {X 502.6885, Y 49.1600, Z -1.3333, A 0.000, B 0.000, C 0.000 }
gfCNCPoint1[14853] = {X 496.2450, Y 49.1600, Z -1.3333, A 0.000, B 0.000, C 0.000 }
gfCNCPoint1[14854] = {X 495.3239, Y 49.0567, Z -1.3333, A 0.000, B 0.000, C 0.000 }
gfCNCPoint1[14855] = {X 494.4485, Y 48.7521, Z -1.3333, A 0.000, B 0.000, C 0.000 }
gfCNCPoint1[14856] = {X 493.6623, Y 48.2612, Z -1.3333, A 0.000, B 0.000, C 0.000 }
gfCNCPoint1[14857] = {X 493.0043, Y 47.6084, Z -1.3333, A 0.000, B 0.000, C 0.000 }
gfCNCPoint1[14858] = {X 492.5072, Y 46.8261, Z -1.3333, A 0.000, B 0.000, C 0.000 }
gfCNCPoint1[14859] = {X 492.1957, Y 45.9531, Z -1.3333, A 0.000, B 0.000, C 0.000 }
gfCNCPoint1[14860] = {X 492.0852, Y 45.0328, Z -1.3333, A 0.000, B 0.000, C 0.000 }
gfCNCPoint1[14861] = {X 492.0854, Y 44.1516, Z -1.3333, A 0.000, B 0.000, C 0.000 }
gfCNCPoint1[14862] = {X 492.1960, Y 43.2545, Z -1.3333, A 0.000, B 0.000, C 0.000 }
gfCNCPoint1[14863] = {X 492.4976, Y 42.4026, Z -1.3333, A 0.000, B 0.000, C 0.000 }
gfCNCPoint1[14864] = {X 492.9762, Y 41.6358, Z -1.3333, A 0.000, B 0.000, C 0.000 }
gfCNCPoint1[14865] = {X 493.6090, Y 40.9906, Z -1.3333, A 0.000, B 0.000, C 0.000 }
gfCNCPoint1[14866] = {X 493.6090, Y 34.3138, Z -1.3333, A 0.000, B 0.000, C 0.000 }
gfCNCPoint1[14867] = {X 490.6255, Y 34.3138, Z -1.3333, A 0.000, B 0.000, C 0.000 }
gfCNCPoint1[14868] = {X 486.2645, Y 42.8059, Z -1.3333, A 0.000, B 0.000, C 0.000 }
gfCNCPoint1[14869] = {X 486.2941, Y 42.8829, Z -1.3333, A 0.000, B 0.000, C 0.000 }
gfCNCPoint1[14870] = {X 486.4534, Y 43.5185, Z -1.3333, A 0.000, B 0.000, C 0.000 }
gfCNCPoint1[14871] = {X 486.5108, Y 44.1713, Z -1.3333, A 0.000, B 0.000, C 0.000 }
gfCNCPoint1[14872] = {X 486.5110, Y 45.0000, Z -1.3333, A 0.000, B 0.000, C 0.000 }
gfCNCPoint1[14873] = {X 486.4067, Y 45.9257, Z -1.3333, A 0.000, B 0.000, C 0.000 }
gfCNCPoint1[14874] = {X 486.0990, Y 46.8050, Z -1.3333, A 0.000, B 0.000, C 0.000 }
gfCNCPoint1[14875] = {X 485.6034, Y 47.5937, Z -1.3333, A 0.000, B 0.000, C 0.000 }
gfCNCPoint1[14876] = {X 484.9447, Y 48.2524, Z -1.3333, A 0.000, B 0.000, C 0.000 }
gfCNCPoint1[14877] = {X 484.1560, Y 48.7480, Z -1.3333, A 0.000, B 0.000, C 0.000 }
gfCNCPoint1[14878] = {X 483.2767, Y 49.0557, Z -1.3333, A 0.000, B 0.000, C 0.000 }
gfCNCPoint1[14879] = {X 482.3510, Y 49.1600, Z -1.3333, A 0.000, B 0.000, C 0.000 }
gfCNCPoint1[14880] = {X 475.7650, Y 49.1600, Z -1.3333, A 0.000, B 0.000, C 0.000 }
gfCNCPoint1[14881] = {X 474.8393, Y 49.0557, Z -1.3333, A 0.000, B 0.000, C 0.000 }
gfCNCPoint1[14882] = {X 473.9600, Y 48.7480, Z -1.3333, A 0.000, B 0.000, C 0.000 }
gfCNCPoint1[14883] = {X 473.1713, Y 48.2524, Z -1.3333, A 0.000, B 0.000, C 0.000 }
gfCNCPoint1[14884] = {X 472.5126, Y 47.5937, Z -1.3333, A 0.000, B 0.000, C 0.000 }
gfCNCPoint1[14885] = {X 472.0169, Y 46.8050, Z -1.3333, A 0.000, B 0.000, C 0.000 }
gfCNCPoint1[14886] = {X 471.7093, Y 45.9257, Z -1.3333, A 0.000, B 0.000, C 0.000 }
gfCNCPoint1[14887] = {X 471.6050, Y 45.0000, Z -1.3333, A 0.000, B 0.000, C 0.000 }
gfCNCPoint1[14888] = {X 471.6054, Y 44.1516, Z -1.3333, A 0.000, B 0.000, C 0.000 }
gfCNCPoint1[14889] = {X 471.7016, Y 43.3174, Z -1.3333, A 0.000, B 0.000, C 0.000 }
gfCNCPoint1[14890] = {X 471.9634, Y 42.5195, Z -1.3333, A 0.000, B 0.000, C 0.000 }
gfCNCPoint1[14891] = {X 472.3801, Y 41.7905, Z -1.3333, A 0.000, B 0.000, C 0.000 }
gfCNCPoint1[14892] = {X 472.9347, Y 41.1600, Z -1.3333, A 0.000, B 0.000, C 0.000 }
gfCNCPoint1[14893] = {X 473.6046, Y 40.6537, Z -1.3333, A 0.000, B 0.000, C 0.000 }
gfCNCPoint1[14894] = {X 474.3626, Y 40.2923, Z -1.3333, A 0.000, B 0.000, C 0.000 }
gfCNCPoint1[14895] = {X 478.4444, Y 32.3026, Z -1.3333, A 0.000, B 0.000, C 0.000 }
gfCNCPoint1[14896] = {X 477.1677, Y 31.4482, Z -1.3333, A 0.000, B 0.000, C 0.000 }
gfCNCPoint1[14897] = {X 476.0187, Y 30.4287, Z -1.3333, A 0.000, B 0.000, C 0.000 }
gfCNCPoint1[14898] = {X 475.0183, Y 29.2629, Z -1.3333, A 0.000, B 0.000, C 0.000 }
gfCNCPoint1[14899] = {X 474.1851, Y 27.9723, Z -1.3333, A 0.000, B 0.000, C 0.000 }
gfCNCPoint1[14900] = {X 473.5345, Y 26.5807, Z -1.3333, A 0.000, B 0.000, C 0.000 }
gfCNCPoint1[14901] = {X 473.0784, Y 25.1138, Z -1.3333, A 0.000, B 0.000, C 0.000 }
gfCNCPoint1[14902] = {X 472.7672, Y 23.4468, Z -1.3333, A 0.000, B 0.000, C 0.000 }
gfCNCPoint1[14903] = {X 472.6280, Y 21.7567, Z -1.3333, A 0.000, B 0.000, C 0.000 }
gfCNCPoint1[14904] = {X 472.6624, Y 20.0612, Z -1.3333, A 0.000, B 0.000, C 0.000 }
gfCNCPoint1[14905] = {X 472.8699, Y 18.3781, Z -1.3333, A 0.000, B 0.000, C 0.000 }
gfCNCPoint1[14906] = {X 473.2484, Y 16.7251, Z -1.3333, A 0.000, B 0.000, C 0.000 }
gfCNCPoint1[14907] = {X 473.7842, Y 15.2312, Z -1.3333, A 0.000, B 0.000, C 0.000 }
gfCNCPoint1[14908] = {X 474.5176, Y 13.8238, Z -1.3333, A 0.000, B 0.000, C 0.000 }
gfCNCPoint1[14909] = {X 475.4351, Y 12.5289, Z -1.3333, A 0.000, B 0.000, C 0.000 }
gfCNCPoint1[14910] = {X 476.5197, Y 11.3703, Z -1.3333, A 0.000, B 0.000, C 0.000 }
gfCNCPoint1[14911] = {X 477.7514, Y 10.3695, Z -1.3333, A 0.000, B 0.000, C 0.000 }
gfCNCPoint1[14912] = {X 479.1075, Y 9.5450, Z -1.3333, A 0.000, B 0.000, C 0.000 }
gfCNCPoint1[14913] = {X 480.5628, Y 8.9120, Z -1.3333, A 0.000, B 0.000, C 0.000 }
gfCNCPoint1[14914] = {X 482.0905, Y 8.4822, Z -1.3333, A 0.000, B 0.000, C 0.000 }
gfCNCPoint1[14915] = {X 484.1725, Y 8.1583, Z -1.3333, A 0.000, B 0.000, C 0.000 }
gfCNCPoint1[14916] = {X 486.2764, Y 8.0441, Z -1.3333, A 0.000, B 0.000, C 0.000 }
gfCNCPoint1[14917] = {X 486.9693, Y 8.0319, Z -1.3333, A 0.000, B 0.000, C 0.000 }
gfCNCPoint1[14918] = {X 492.3824, Y 8.0319, Z -1.3333, A 0.000, B 0.000, C 0.000 }
gfCNCPoint1[14919] = {X 492.3824, Y 4.0319, Z -1.3333, A 0.000, B 0.000, C 0.000 }
gfCNCPoint1[14920] = {X 492.3824, Y 8.1119, Z -1.3333, A 0.000, B 0.000, C 0.000 }
gfCNCPoint1[14921] = {X 502.2056, Y 8.1119, Z -1.3333, A 0.000, B 0.000, C 0.000 }
gfCNCPoint1[14922] = {X 502.7354, Y 8.1160, Z -1.3333, A 0.000, B 0.000, C 0.000 }
gfCNCPoint1[14923] = {X 503.6347, Y 8.2240, Z -1.3333, A 0.000, B 0.000, C 0.000 }
gfCNCPoint1[14924] = {X 504.4877, Y 8.5284, Z -1.3333, A 0.000, B 0.000, C 0.000 }
gfCNCPoint1[14925] = {X 505.2522, Y 9.0141, Z -1.3333, A 0.000, B 0.000, C 0.000 }
gfCNCPoint1[14926] = {X 505.8901, Y 9.6570, Z -1.3333, A 0.000, B 0.000, C 0.000 }
gfCNCPoint1[14927] = {X 506.3699, Y 10.4253, Z -1.3333, A 0.000, B 0.000, C 0.000 }
gfCNCPoint1[14928] = {X 506.6676, Y 11.2807, Z -1.3333, A 0.000, B 0.000, C 0.000 }
gfCNCPoint1[14929] = {X 506.7685, Y 12.1807, Z -1.3333, A 0.000, B 0.000, C 0.000 }
gfCNCPoint1[14930] = {X 506.7685, Y 12.9781, Z -1.3333, A 0.000, B 0.000, C 0.000 }
gfCNCPoint1[14931] = {X 506.6667, Y 13.8836, Z -1.3333, A 0.000, B 0.000, C 0.000 }
gfCNCPoint1[14932] = {X 506.3665, Y 14.7439, Z -1.3333, A 0.000, B 0.000, C 0.000 }
gfCNCPoint1[14933] = {X 505.8829, Y 15.5161, Z -1.3333, A 0.000, B 0.000, C 0.000 }
gfCNCPoint1[14934] = {X 505.2400, Y 16.1618, Z -1.3333, A 0.000, B 0.000, C 0.000 }
gfCNCPoint1[14935] = {X 505.2399, Y 41.0273, Z -1.3333, A 0.000, B 0.000, C 0.000 }
gfCNCPoint1[14936] = {X 505.3177, Y 41.0889, Z -1.3333, A 0.000, B 0.000, C 0.000 }
gfCNCPoint1[14937] = {X 505.9239, Y 41.7232, Z -1.3333, A 0.000, B 0.000, C 0.000 }
gfCNCPoint1[14938] = {X 506.3805, Y 42.4724, Z -1.3333, A 0.000, B 0.000, C 0.000 }
gfCNCPoint1[14939] = {X 506.6664, Y 43.3019, Z -1.3333, A 0.000, B 0.000, C 0.000 }
gfCNCPoint1[14940] = {X 506.7683, Y 44.1734, Z -1.3333, A 0.000, B 0.000, C 0.000 }
gfCNCPoint1[14941] = {X 506.7685, Y 45.0000, Z -1.3333, A 0.000, B 0.000, C 0.000 }
gfCNCPoint1[14942] = {X 506.6662, Y 45.9079, Z -1.3333, A 0.000, B 0.000, C 0.000 }
gfCNCPoint1[14943] = {X 506.3644, Y 46.7702, Z -1.3333, A 0.000, B 0.000, C 0.000 }
gfCNCPoint1[14944] = {X 505.8784, Y 47.5438, Z -1.3333, A 0.000, B 0.000, C 0.000 }
gfCNCPoint1[14945] = {X 505.2323, Y 48.1899, Z -1.3333, A 0.000, B 0.000, C 0.000 }
gfCNCPoint1[14946] = {X 504.4587, Y 48.6760, Z -1.3333, A 0.000, B 0.000, C 0.000 }
gfCNCPoint1[14947] = {X 503.5964, Y 48.9777, Z -1.3333, A 0.000, B 0.000, C 0.000 }
gfCNCPoint1[14948] = {X 502.6885, Y 49.0800, Z -1.3333, A 0.000, B 0.000, C 0.000 }
gfCNCPoint1[14949] = {X 496.2450, Y 49.0800, Z -1.3333, A 0.000, B 0.000, C 0.000 }
gfCNCPoint1[14950] = {X 495.3416, Y 48.9787, Z -1.3333, A 0.000, B 0.000, C 0.000 }
gfCNCPoint1[14951] = {X 494.4831, Y 48.6799, Z -1.3333, A 0.000, B 0.000, C 0.000 }
gfCNCPoint1[14952] = {X 493.7120, Y 48.1985, Z -1.3333, A 0.000, B 0.000, C 0.000 }
gfCNCPoint1[14953] = {X 493.0667, Y 47.5582, Z -1.3333, A 0.000, B 0.000, C 0.000 }
gfCNCPoint1[14954] = {X 492.5791, Y 46.7909, Z -1.3333, A 0.000, B 0.000, C 0.000 }
gfCNCPoint1[14955] = {X 492.2736, Y 45.9348, Z -1.3333, A 0.000, B 0.000, C 0.000 }
gfCNCPoint1[14956] = {X 492.1652, Y 45.0322, Z -1.3333, A 0.000, B 0.000, C 0.000 }
gfCNCPoint1[14957] = {X 492.1654, Y 44.1527, Z -1.3333, A 0.000, B 0.000, C 0.000 }
gfCNCPoint1[14958] = {X 492.2760, Y 43.2637, Z -1.3333, A 0.000, B 0.000, C 0.000 }
gfCNCPoint1[14959] = {X 492.5779, Y 42.4203, Z -1.3333, A 0.000, B 0.000, C 0.000 }
gfCNCPoint1[14960] = {X 493.0566, Y 41.6631, Z -1.3333, A 0.000, B 0.000, C 0.000 }
gfCNCPoint1[14961] = {X 493.6890, Y 41.0287, Z -1.3333, A 0.000, B 0.000, C 0.000 }
gfCNCPoint1[14962] = {X 493.6890, Y 34.2338, Z -1.3333, A 0.000, B 0.000, C 0.000 }
gfCNCPoint1[14963] = {X 490.5766, Y 34.2338, Z -1.3333, A 0.000, B 0.000, C 0.000 }
gfCNCPoint1[14964] = {X 486.1770, Y 42.8012, Z -1.3333, A 0.000, B 0.000, C 0.000 }
gfCNCPoint1[14965] = {X 486.2188, Y 42.9100, Z -1.3333, A 0.000, B 0.000, C 0.000 }
gfCNCPoint1[14966] = {X 486.3746, Y 43.5326, Z -1.3333, A 0.000, B 0.000, C 0.000 }
gfCNCPoint1[14967] = {X 486.4309, Y 44.1720, Z -1.3333, A 0.000, B 0.000, C 0.000 }
gfCNCPoint1[14968] = {X 486.4310, Y 45.0000, Z -1.3333, A 0.000, B 0.000, C 0.000 }
gfCNCPoint1[14969] = {X 486.3287, Y 45.9079, Z -1.3333, A 0.000, B 0.000, C 0.000 }
gfCNCPoint1[14970] = {X 486.0270, Y 46.7702, Z -1.3333, A 0.000, B 0.000, C 0.000 }
gfCNCPoint1[14971] = {X 485.5409, Y 47.5438, Z -1.3333, A 0.000, B 0.000, C 0.000 }
gfCNCPoint1[14972] = {X 484.8949, Y 48.1899, Z -1.3333, A 0.000, B 0.000, C 0.000 }
gfCNCPoint1[14973] = {X 484.1213, Y 48.6760, Z -1.3333, A 0.000, B 0.000, C 0.000 }
gfCNCPoint1[14974] = {X 483.2589, Y 48.9777, Z -1.3333, A 0.000, B 0.000, C 0.000 }
gfCNCPoint1[14975] = {X 482.3510, Y 49.0800, Z -1.3333, A 0.000, B 0.000, C 0.000 }
gfCNCPoint1[14976] = {X 475.7650, Y 49.0800, Z -1.3333, A 0.000, B 0.000, C 0.000 }
gfCNCPoint1[14977] = {X 474.8571, Y 48.9777, Z -1.3333, A 0.000, B 0.000, C 0.000 }
gfCNCPoint1[14978] = {X 473.9947, Y 48.6760, Z -1.3333, A 0.000, B 0.000, C 0.000 }
gfCNCPoint1[14979] = {X 473.2211, Y 48.1899, Z -1.3333, A 0.000, B 0.000, C 0.000 }
gfCNCPoint1[14980] = {X 472.5751, Y 47.5438, Z -1.3333, A 0.000, B 0.000, C 0.000 }
gfCNCPoint1[14981] = {X 472.0890, Y 46.7702, Z -1.3333, A 0.000, B 0.000, C 0.000 }
gfCNCPoint1[14982] = {X 471.7873, Y 45.9079, Z -1.3333, A 0.000, B 0.000, C 0.000 }
gfCNCPoint1[14983] = {X 471.6850, Y 45.0000, Z -1.3333, A 0.000, B 0.000, C 0.000 }
gfCNCPoint1[14984] = {X 471.6853, Y 44.1527, Z -1.3333, A 0.000, B 0.000, C 0.000 }
gfCNCPoint1[14985] = {X 471.7809, Y 43.3294, Z -1.3333, A 0.000, B 0.000, C 0.000 }
gfCNCPoint1[14986] = {X 472.0408, Y 42.5424, Z -1.3333, A 0.000, B 0.000, C 0.000 }
gfCNCPoint1[14987] = {X 472.4544, Y 41.8242, Z -1.3333, A 0.000, B 0.000, C 0.000 }
gfCNCPoint1[14988] = {X 473.0046, Y 41.2044, Z -1.3333, A 0.000, B 0.000, C 0.000 }
gfCNCPoint1[14989] = {X 473.6687, Y 40.7085, Z -1.3333, A 0.000, B 0.000, C 0.000 }
gfCNCPoint1[14990] = {X 474.4193, Y 40.3571, Z -1.3333, A 0.000, B 0.000, C 0.000 }
gfCNCPoint1[14991] = {X 478.5504, Y 32.2709, Z -1.3333, A 0.000, B 0.000, C 0.000 }
gfCNCPoint1[14992] = {X 477.2669, Y 31.4235, Z -1.3333, A 0.000, B 0.000, C 0.000 }
gfCNCPoint1[14993] = {X 476.1113, Y 30.4086, Z -1.3333, A 0.000, B 0.000, C 0.000 }
gfCNCPoint1[14994] = {X 475.1052, Y 29.2454, Z -1.3333, A 0.000, B 0.000, C 0.000 }
gfCNCPoint1[14995] = {X 474.2674, Y 27.9557, Z -1.3333, A 0.000, B 0.000, C 0.000 }
gfCNCPoint1[14996] = {X 473.6136, Y 26.5635, Z -1.3333, A 0.000, B 0.000, C 0.000 }
gfCNCPoint1[14997] = {X 473.1562, Y 25.0952, Z -1.3333, A 0.000, B 0.000, C 0.000 }
gfCNCPoint1[14998] = {X 472.8465, Y 23.4362, Z -1.3333, A 0.000, B 0.000, C 0.000 }
gfCNCPoint1[14999] = {X 472.7080, Y 21.7542, Z -1.3333, A 0.000, B 0.000, C 0.000 }
gfCNCPoint1[15000] = {X 472.7422, Y 20.0669, Z -1.3333, A 0.000, B 0.000, C 0.000 }
gfCNCPoint1[15001] = {X 472.9487, Y 18.3920, Z -1.3333, A 0.000, B 0.000, C 0.000 }
gfCNCPoint1[15002] = {X 473.3254, Y 16.7469, Z -1.3333, A 0.000, B 0.000, C 0.000 }
gfCNCPoint1[15003] = {X 473.8575, Y 15.2633, Z -1.3333, A 0.000, B 0.000, C 0.000 }
gfCNCPoint1[15004] = {X 474.5859, Y 13.8655, Z -1.3333, A 0.000, B 0.000, C 0.000 }
gfCNCPoint1[15005] = {X 475.4971, Y 12.5795, Z -1.3333, A 0.000, B 0.000, C 0.000 }
gfCNCPoint1[15006] = {X 476.5743, Y 11.4288, Z -1.3333, A 0.000, B 0.000, C 0.000 }
gfCNCPoint1[15007] = {X 477.7976, Y 10.4349, Z -1.3333, A 0.000, B 0.000, C 0.000 }
gfCNCPoint1[15008] = {X 479.1443, Y 9.6160, Z -1.3333, A 0.000, B 0.000, C 0.000 }
gfCNCPoint1[15009] = {X 480.5897, Y 8.9874, Z -1.3333, A 0.000, B 0.000, C 0.000 }
gfCNCPoint1[15010] = {X 482.1069, Y 8.5605, Z -1.3333, A 0.000, B 0.000, C 0.000 }
gfCNCPoint1[15011] = {X 484.1812, Y 8.2378, Z -1.3333, A 0.000, B 0.000, C 0.000 }
gfCNCPoint1[15012] = {X 486.2773, Y 8.1241, Z -1.3333, A 0.000, B 0.000, C 0.000 }
gfCNCPoint1[15013] = {X 486.9700, Y 8.1119, Z -1.3333, A 0.000, B 0.000, C 0.000 }
gfCNCPoint1[15014] = {X 492.3824, Y 8.1119, Z -1.3333, A 0.000, B 0.000, C 0.000 }
gfCNCPoint1[15015] = {X 492.3824, Y 4.1119, Z -1.3333, A 0.000, B 0.000, C 0.000 }
gfCNCPoint1[15016] = {X 492.3824, Y 8.1919, Z -1.3333, A 0.000, B 0.000, C 0.000 }
gfCNCPoint1[15017] = {X 502.2053, Y 8.1919, Z -1.3333, A 0.000, B 0.000, C 0.000 }
gfCNCPoint1[15018] = {X 502.7348, Y 8.1960, Z -1.3333, A 0.000, B 0.000, C 0.000 }
gfCNCPoint1[15019] = {X 503.6164, Y 8.3018, Z -1.3333, A 0.000, B 0.000, C 0.000 }
gfCNCPoint1[15020] = {X 504.4526, Y 8.6002, Z -1.3333, A 0.000, B 0.000, C 0.000 }
gfCNCPoint1[15021] = {X 505.2020, Y 9.0764, Z -1.3333, A 0.000, B 0.000, C 0.000 }
gfCNCPoint1[15022] = {X 505.8274, Y 9.7067, Z -1.3333, A 0.000, B 0.000, C 0.000 }
gfCNCPoint1[15023] = {X 506.2977, Y 10.4598, Z -1.3333, A 0.000, B 0.000, C 0.000 }
gfCNCPoint1[15024] = {X 506.5896, Y 11.2984, Z -1.3333, A 0.000, B 0.000, C 0.000 }
gfCNCPoint1[15025] = {X 506.6885, Y 12.1807, Z -1.3333, A 0.000, B 0.000, C 0.000 }
gfCNCPoint1[15026] = {X 506.6883, Y 13.0192, Z -1.3333, A 0.000, B 0.000, C 0.000 }
gfCNCPoint1[15027] = {X 506.5796, Y 13.9052, Z -1.3333, A 0.000, B 0.000, C 0.000 }
gfCNCPoint1[15028] = {X 506.2771, Y 14.7449, Z -1.3333, A 0.000, B 0.000, C 0.000 }
gfCNCPoint1[15029] = {X 505.7959, Y 15.4968, Z -1.3333, A 0.000, B 0.000, C 0.000 }
gfCNCPoint1[15030] = {X 505.1600, Y 16.1231, Z -1.3333, A 0.000, B 0.000, C 0.000 }
gfCNCPoint1[15031] = {X 505.1599, Y 41.0660, Z -1.3333, A 0.000, B 0.000, C 0.000 }
gfCNCPoint1[15032] = {X 505.2989, Y 41.1780, Z -1.3333, A 0.000, B 0.000, C 0.000 }
gfCNCPoint1[15033] = {X 505.8853, Y 41.8045, Z -1.3333, A 0.000, B 0.000, C 0.000 }
gfCNCPoint1[15034] = {X 506.3246, Y 42.5418, Z -1.3333, A 0.000, B 0.000, C 0.000 }
gfCNCPoint1[15035] = {X 506.5965, Y 43.3557, Z -1.3333, A 0.000, B 0.000, C 0.000 }
gfCNCPoint1[15036] = {X 506.6885, Y 44.2089, Z -1.3333, A 0.000, B 0.000, C 0.000 }
gfCNCPoint1[15037] = {X 506.6885, Y 45.0000, Z -1.3333, A 0.000, B 0.000, C 0.000 }
gfCNCPoint1[15038] = {X 506.5882, Y 45.8901, Z -1.3333, A 0.000, B 0.000, C 0.000 }
gfCNCPoint1[15039] = {X 506.2924, Y 46.7355, Z -1.3333, A 0.000, B 0.000, C 0.000 }
gfCNCPoint1[15040] = {X 505.8158, Y 47.4940, Z -1.3333, A 0.000, B 0.000, C 0.000 }
gfCNCPoint1[15041] = {X 505.1825, Y 48.1273, Z -1.3333, A 0.000, B 0.000, C 0.000 }
gfCNCPoint1[15042] = {X 504.4240, Y 48.6039, Z -1.3333, A 0.000, B 0.000, C 0.000 }
gfCNCPoint1[15043] = {X 503.5786, Y 48.8997, Z -1.3333, A 0.000, B 0.000, C 0.000 }
gfCNCPoint1[15044] = {X 502.6885, Y 49.0000, Z -1.3333, A 0.000, B 0.000, C 0.000 }
gfCNCPoint1[15045] = {X 496.2450, Y 49.0000, Z -1.3333, A 0.000, B 0.000, C 0.000 }
gfCNCPoint1[15046] = {X 495.3549, Y 48.8997, Z -1.3333, A 0.000, B 0.000, C 0.000 }
gfCNCPoint1[15047] = {X 494.5095, Y 48.6039, Z -1.3333, A 0.000, B 0.000, C 0.000 }
gfCNCPoint1[15048] = {X 493.7510, Y 48.1273, Z -1.3333, A 0.000, B 0.000, C 0.000 }
gfCNCPoint1[15049] = {X 493.1177, Y 47.4939, Z -1.3333, A 0.000, B 0.000, C 0.000 }
gfCNCPoint1[15050] = {X 492.6411, Y 46.7355, Z -1.3333, A 0.000, B 0.000, C 0.000 }
gfCNCPoint1[15051] = {X 492.3453, Y 45.8900, Z -1.3333, A 0.000, B 0.000, C 0.000 }
gfCNCPoint1[15052] = {X 492.2450, Y 44.9999, Z -1.3333, A 0.000, B 0.000, C 0.000 }
gfCNCPoint1[15053] = {X 492.2454, Y 44.1538, Z -1.3333, A 0.000, B 0.000, C 0.000 }
gfCNCPoint1[15054] = {X 492.3560, Y 43.2730, Z -1.3333, A 0.000, B 0.000, C 0.000 }
gfCNCPoint1[15055] = {X 492.6582, Y 42.4382, Z -1.3333, A 0.000, B 0.000, C 0.000 }
gfCNCPoint1[15056] = {X 493.1371, Y 41.6907, Z -1.3333, A 0.000, B 0.000, C 0.000 }
gfCNCPoint1[15057] = {X 493.7690, Y 41.0672, Z -1.3333, A 0.000, B 0.000, C 0.000 }
gfCNCPoint1[15058] = {X 493.7690, Y 34.1538, Z -1.3333, A 0.000, B 0.000, C 0.000 }
gfCNCPoint1[15059] = {X 490.7720, Y 34.1538, Z -1.3333, A 0.000, B 0.000, C 0.000 }
gfCNCPoint1[15060] = {X 490.5295, Y 34.1504, Z -1.3333, A 0.000, B 0.000, C 0.000 }
gfCNCPoint1[15061] = {X 486.0895, Y 42.7965, Z -1.3333, A 0.000, B 0.000, C 0.000 }
gfCNCPoint1[15062] = {X 486.1469, Y 42.9473, Z -1.3333, A 0.000, B 0.000, C 0.000 }
gfCNCPoint1[15063] = {X 486.2997, Y 43.5699, Z -1.3333, A 0.000, B 0.000, C 0.000 }
gfCNCPoint1[15064] = {X 486.3510, Y 44.2089, Z -1.3333, A 0.000, B 0.000, C 0.000 }
gfCNCPoint1[15065] = {X 486.3510, Y 45.0000, Z -1.3333, A 0.000, B 0.000, C 0.000 }
gfCNCPoint1[15066] = {X 486.2507, Y 45.8901, Z -1.3333, A 0.000, B 0.000, C 0.000 }
gfCNCPoint1[15067] = {X 485.9549, Y 46.7355, Z -1.3333, A 0.000, B 0.000, C 0.000 }
gfCNCPoint1[15068] = {X 485.4783, Y 47.4940, Z -1.3333, A 0.000, B 0.000, C 0.000 }
gfCNCPoint1[15069] = {X 484.8450, Y 48.1273, Z -1.3333, A 0.000, B 0.000, C 0.000 }
gfCNCPoint1[15070] = {X 484.0866, Y 48.6039, Z -1.3333, A 0.000, B 0.000, C 0.000 }
gfCNCPoint1[15071] = {X 483.2411, Y 48.8997, Z -1.3333, A 0.000, B 0.000, C 0.000 }
gfCNCPoint1[15072] = {X 482.3510, Y 49.0000, Z -1.3333, A 0.000, B 0.000, C 0.000 }
gfCNCPoint1[15073] = {X 475.7650, Y 49.0000, Z -1.3333, A 0.000, B 0.000, C 0.000 }
gfCNCPoint1[15074] = {X 474.8749, Y 48.8997, Z -1.3333, A 0.000, B 0.000, C 0.000 }
gfCNCPoint1[15075] = {X 474.0294, Y 48.6039, Z -1.3333, A 0.000, B 0.000, C 0.000 }
gfCNCPoint1[15076] = {X 473.2710, Y 48.1273, Z -1.3333, A 0.000, B 0.000, C 0.000 }
gfCNCPoint1[15077] = {X 472.6376, Y 47.4940, Z -1.3333, A 0.000, B 0.000, C 0.000 }
gfCNCPoint1[15078] = {X 472.1611, Y 46.7355, Z -1.3333, A 0.000, B 0.000, C 0.000 }
gfCNCPoint1[15079] = {X 471.8652, Y 45.8901, Z -1.3333, A 0.000, B 0.000, C 0.000 }
gfCNCPoint1[15080] = {X 471.7650, Y 45.0000, Z -1.3333, A 0.000, B 0.000, C 0.000 }
gfCNCPoint1[15081] = {X 471.7653, Y 44.1538, Z -1.3333, A 0.000, B 0.000, C 0.000 }
gfCNCPoint1[15082] = {X 471.8601, Y 43.3414, Z -1.3333, A 0.000, B 0.000, C 0.000 }
gfCNCPoint1[15083] = {X 472.1182, Y 42.5654, Z -1.3333, A 0.000, B 0.000, C 0.000 }
gfCNCPoint1[15084] = {X 472.5286, Y 41.8580, Z -1.3333, A 0.000, B 0.000, C 0.000 }
gfCNCPoint1[15085] = {X 473.0744, Y 41.2489, Z -1.3333, A 0.000, B 0.000, C 0.000 }
gfCNCPoint1[15086] = {X 473.7327, Y 40.7635, Z -1.3333, A 0.000, B 0.000, C 0.000 }
gfCNCPoint1[15087] = {X 474.4759, Y 40.4222, Z -1.3333, A 0.000, B 0.000, C 0.000 }
gfCNCPoint1[15088] = {X 478.6566, Y 32.2388, Z -1.3333, A 0.000, B 0.000, C 0.000 }
gfCNCPoint1[15089] = {X 477.3664, Y 31.3985, Z -1.3333, A 0.000, B 0.000, C 0.000 }
gfCNCPoint1[15090] = {X 476.2042, Y 30.3884, Z -1.3333, A 0.000, B 0.000, C 0.000 }
gfCNCPoint1[15091] = {X 475.1922, Y 29.2279, Z -1.3333, A 0.000, B 0.000, C 0.000 }
gfCNCPoint1[15092] = {X 474.3497, Y 27.9390, Z -1.3333, A 0.000, B 0.000, C 0.000 }
gfCNCPoint1[15093] = {X 473.6928, Y 26.5464, Z -1.3333, A 0.000, B 0.000, C 0.000 }
gfCNCPoint1[15094] = {X 473.2340, Y 25.0766, Z -1.3333, A 0.000, B 0.000, C 0.000 }
gfCNCPoint1[15095] = {X 472.9258, Y 23.4256, Z -1.3333, A 0.000, B 0.000, C 0.000 }
gfCNCPoint1[15096] = {X 472.7879, Y 21.7518, Z -1.3333, A 0.000, B 0.000, C 0.000 }
gfCNCPoint1[15097] = {X 472.8220, Y 20.0727, Z -1.3333, A 0.000, B 0.000, C 0.000 }
gfCNCPoint1[15098] = {X 473.0275, Y 18.4058, Z -1.3333, A 0.000, B 0.000, C 0.000 }
gfCNCPoint1[15099] = {X 473.4024, Y 16.7687, Z -1.3333, A 0.000, B 0.000, C 0.000 }
gfCNCPoint1[15100] = {X 473.9308, Y 15.2954, Z -1.3333, A 0.000, B 0.000, C 0.000 }
gfCNCPoint1[15101] = {X 474.6542, Y 13.9072, Z -1.3333, A 0.000, B 0.000, C 0.000 }
gfCNCPoint1[15102] = {X 475.5591, Y 12.6300, Z -1.3333, A 0.000, B 0.000, C 0.000 }
gfCNCPoint1[15103] = {X 476.6288, Y 11.4874, Z -1.3333, A 0.000, B 0.000, C 0.000 }
gfCNCPoint1[15104] = {X 477.8437, Y 10.5003, Z -1.3333, A 0.000, B 0.000, C 0.000 }
gfCNCPoint1[15105] = {X 479.1811, Y 9.6871, Z -1.3333, A 0.000, B 0.000, C 0.000 }
gfCNCPoint1[15106] = {X 480.6165, Y 9.0627, Z -1.3333, A 0.000, B 0.000, C 0.000 }
gfCNCPoint1[15107] = {X 482.1233, Y 8.6388, Z -1.3333, A 0.000, B 0.000, C 0.000 }
gfCNCPoint1[15108] = {X 484.1898, Y 8.3173, Z -1.3333, A 0.000, B 0.000, C 0.000 }
gfCNCPoint1[15109] = {X 486.2782, Y 8.2041, Z -1.3333, A 0.000, B 0.000, C 0.000 }
gfCNCPoint1[15110] = {X 486.9707, Y 8.1919, Z -1.3333, A 0.000, B 0.000, C 0.000 }
gfCNCPoint1[15111] = {X 492.3824, Y 8.1919, Z -1.3333, A 0.000, B 0.000, C 0.000 }
gfCNCPoint1[15112] = {X 492.3824, Y 4.1119, Z -1.3333, A 0.000, B 0.000, C 0.000 }
gfCNCPoint1[15113] = {X 492.3824, Y 4.1119, Z 1.6667, A 0.000, B 0.000, C 0.000 }
gfCNCPoint1[15114] = {X 492.3824, Y 4.1119, Z 11.0000, A 0.000, B 0.000, C 0.000 }
gfCNCPoint1[15115] = {X 533.9642, Y 3.7916, Z 11.0000, A 0.000, B 0.000, C 0.000 }
gfCNCPoint1[15116] = {X 533.9642, Y 3.7916, Z 1.6667, A 0.000, B 0.000, C 0.000 }
gfCNCPoint1[15117] = {X 533.9642, Y 3.7916, Z -1.3333, A 0.000, B 0.000, C 0.000 }
gfCNCPoint1[15118] = {X 533.9641, Y 7.8716, Z -1.3333, A 0.000, B 0.000, C 0.000 }
gfCNCPoint1[15119] = {X 543.7499, Y 7.8719, Z -1.3333, A 0.000, B 0.000, C 0.000 }
gfCNCPoint1[15120] = {X 544.7299, Y 7.9574, Z -1.3333, A 0.000, B 0.000, C 0.000 }
gfCNCPoint1[15121] = {X 545.6653, Y 8.2622, Z -1.3333, A 0.000, B 0.000, C 0.000 }
gfCNCPoint1[15122] = {X 546.5075, Y 8.7704, Z -1.3333, A 0.000, B 0.000, C 0.000 }
gfCNCPoint1[15123] = {X 547.2132, Y 9.4559, Z -1.3333, A 0.000, B 0.000, C 0.000 }
gfCNCPoint1[15124] = {X 547.7457, Y 10.2830, Z -1.3333, A 0.000, B 0.000, C 0.000 }
gfCNCPoint1[15125] = {X 548.0775, Y 11.2091, Z -1.3333, A 0.000, B 0.000, C 0.000 }
gfCNCPoint1[15126] = {X 548.1914, Y 12.1862, Z -1.3333, A 0.000, B 0.000, C 0.000 }
gfCNCPoint1[15127] = {X 548.1912, Y 13.0225, Z -1.3333, A 0.000, B 0.000, C 0.000 }
gfCNCPoint1[15128] = {X 548.0827, Y 13.9409, Z -1.3333, A 0.000, B 0.000, C 0.000 }
gfCNCPoint1[15129] = {X 547.7811, Y 14.8152, Z -1.3333, A 0.000, B 0.000, C 0.000 }
gfCNCPoint1[15130] = {X 547.3004, Y 15.6052, Z -1.3333, A 0.000, B 0.000, C 0.000 }
gfCNCPoint1[15131] = {X 546.6626, Y 16.2748, Z -1.3333, A 0.000, B 0.000, C 0.000 }
gfCNCPoint1[15132] = {X 546.6628, Y 40.9129, Z -1.3333, A 0.000, B 0.000, C 0.000 }
gfCNCPoint1[15133] = {X 546.6853, Y 40.9309, Z -1.3333, A 0.000, B 0.000, C 0.000 }
gfCNCPoint1[15134] = {X 547.3154, Y 41.6008, Z -1.3333, A 0.000, B 0.000, C 0.000 }
gfCNCPoint1[15135] = {X 547.7894, Y 42.3890, Z -1.3333, A 0.000, B 0.000, C 0.000 }
gfCNCPoint1[15136] = {X 548.0859, Y 43.2596, Z -1.3333, A 0.000, B 0.000, C 0.000 }
gfCNCPoint1[15137] = {X 548.1913, Y 44.1733, Z -1.3333, A 0.000, B 0.000, C 0.000 }
gfCNCPoint1[15138] = {X 548.1914, Y 45.0006, Z -1.3333, A 0.000, B 0.000, C 0.000 }
gfCNCPoint1[15139] = {X 548.0775, Y 45.9777, Z -1.3333, A 0.000, B 0.000, C 0.000 }
gfCNCPoint1[15140] = {X 547.7457, Y 46.9038, Z -1.3333, A 0.000, B 0.000, C 0.000 }
gfCNCPoint1[15141] = {X 547.2131, Y 47.7309, Z -1.3333, A 0.000, B 0.000, C 0.000 }
gfCNCPoint1[15142] = {X 546.5075, Y 48.4163, Z -1.3333, A 0.000, B 0.000, C 0.000 }
gfCNCPoint1[15143] = {X 545.6652, Y 48.9244, Z -1.3333, A 0.000, B 0.000, C 0.000 }
gfCNCPoint1[15144] = {X 544.7299, Y 49.2291, Z -1.3333, A 0.000, B 0.000, C 0.000 }
gfCNCPoint1[15145] = {X 543.7499, Y 49.3146, Z -1.3333, A 0.000, B 0.000, C 0.000 }
gfCNCPoint1[15146] = {X 524.0446, Y 49.3152, Z -1.3333, A 0.000, B 0.000, C 0.000 }
gfCNCPoint1[15147] = {X 523.4981, Y 49.9491, Z -1.3333, A 0.000, B 0.000, C 0.000 }
gfCNCPoint1[15148] = {X 522.8432, Y 50.4704, Z -1.3333, A 0.000, B 0.000, C 0.000 }
gfCNCPoint1[15149] = {X 522.1028, Y 50.8607, Z -1.3333, A 0.000, B 0.000, C 0.000 }
gfCNCPoint1[15150] = {X 521.3027, Y 51.1065, Z -1.3333, A 0.000, B 0.000, C 0.000 }
gfCNCPoint1[15151] = {X 520.4709, Y 51.1991, Z -1.3333, A 0.000, B 0.000, C 0.000 }
gfCNCPoint1[15152] = {X 519.7998, Y 51.1991, Z -1.3333, A 0.000, B 0.000, C 0.000 }
gfCNCPoint1[15153] = {X 518.8385, Y 51.0908, Z -1.3333, A 0.000, B 0.000, C 0.000 }
gfCNCPoint1[15154] = {X 517.9254, Y 50.7713, Z -1.3333, A 0.000, B 0.000, C 0.000 }
gfCNCPoint1[15155] = {X 517.1063, Y 50.2566, Z -1.3333, A 0.000, B 0.000, C 0.000 }
gfCNCPoint1[15156] = {X 516.4223, Y 49.5726, Z -1.3333, A 0.000, B 0.000, C 0.000 }
gfCNCPoint1[15157] = {X 515.9076, Y 48.7535, Z -1.3333, A 0.000, B 0.000, C 0.000 }
gfCNCPoint1[15158] = {X 515.5881, Y 47.8404, Z -1.3333, A 0.000, B 0.000, C 0.000 }
gfCNCPoint1[15159] = {X 515.4798, Y 46.8791, Z -1.3333, A 0.000, B 0.000, C 0.000 }
gfCNCPoint1[15160] = {X 515.4798, Y 39.9011, Z -1.3333, A 0.000, B 0.000, C 0.000 }
gfCNCPoint1[15161] = {X 515.5869, Y 38.9451, Z -1.3333, A 0.000, B 0.000, C 0.000 }
gfCNCPoint1[15162] = {X 515.9029, Y 38.0365, Z -1.3333, A 0.000, B 0.000, C 0.000 }
gfCNCPoint1[15163] = {X 516.4121, Y 37.2204, Z -1.3333, A 0.000, B 0.000, C 0.000 }
gfCNCPoint1[15164] = {X 517.0893, Y 36.5372, Z -1.3333, A 0.000, B 0.000, C 0.000 }
gfCNCPoint1[15165] = {X 517.9010, Y 36.0208, Z -1.3333, A 0.000, B 0.000, C 0.000 }
gfCNCPoint1[15166] = {X 518.8067, Y 35.6968, Z -1.3333, A 0.000, B 0.000, C 0.000 }
gfCNCPoint1[15167] = {X 519.7617, Y 35.5813, Z -1.3333, A 0.000, B 0.000, C 0.000 }
gfCNCPoint1[15168] = {X 520.5269, Y 35.5815, Z -1.3333, A 0.000, B 0.000, C 0.000 }
gfCNCPoint1[15169] = {X 521.3536, Y 35.6728, Z -1.3333, A 0.000, B 0.000, C 0.000 }
gfCNCPoint1[15170] = {X 522.1475, Y 35.9209, Z -1.3333, A 0.000, B 0.000, C 0.000 }
gfCNCPoint1[15171] = {X 522.8792, Y 36.3165, Z -1.3333, A 0.000, B 0.000, C 0.000 }
gfCNCPoint1[15172] = {X 523.5215, Y 36.8450, Z -1.3333, A 0.000, B 0.000, C 0.000 }
gfCNCPoint1[15173] = {X 524.0506, Y 37.4868, Z -1.3333, A 0.000, B 0.000, C 0.000 }
gfCNCPoint1[15174] = {X 534.6319, Y 37.4874, Z -1.3333, A 0.000, B 0.000, C 0.000 }
gfCNCPoint1[15175] = {X 534.6319, Y 33.9645, Z -1.3333, A 0.000, B 0.000, C 0.000 }
gfCNCPoint1[15176] = {X 530.1094, Y 33.9659, Z -1.3333, A 0.000, B 0.000, C 0.000 }
gfCNCPoint1[15177] = {X 529.5772, Y 34.6101, Z -1.3333, A 0.000, B 0.000, C 0.000 }
gfCNCPoint1[15178] = {X 528.9310, Y 35.1398, Z -1.3333, A 0.000, B 0.000, C 0.000 }
gfCNCPoint1[15179] = {X 528.1948, Y 35.5351, Z -1.3333, A 0.000, B 0.000, C 0.000 }
gfCNCPoint1[15180] = {X 527.3964, Y 35.7814, Z -1.3333, A 0.000, B 0.000, C 0.000 }
gfCNCPoint1[15181] = {X 526.5655, Y 35.8693, Z -1.3333, A 0.000, B 0.000, C 0.000 }
gfCNCPoint1[15182] = {X 525.8868, Y 35.8694, Z -1.3333, A 0.000, B 0.000, C 0.000 }
gfCNCPoint1[15183] = {X 524.9255, Y 35.7611, Z -1.3333, A 0.000, B 0.000, C 0.000 }
gfCNCPoint1[15184] = {X 524.0124, Y 35.4416, Z -1.3333, A 0.000, B 0.000, C 0.000 }
gfCNCPoint1[15185] = {X 523.1933, Y 34.9270, Z -1.3333, A 0.000, B 0.000, C 0.000 }
gfCNCPoint1[15186] = {X 522.5092, Y 34.2429, Z -1.3333, A 0.000, B 0.000, C 0.000 }
gfCNCPoint1[15187] = {X 521.9946, Y 33.4238, Z -1.3333, A 0.000, B 0.000, C 0.000 }
gfCNCPoint1[15188] = {X 521.6751, Y 32.5107, Z -1.3333, A 0.000, B 0.000, C 0.000 }
gfCNCPoint1[15189] = {X 521.5668, Y 31.5494, Z -1.3333, A 0.000, B 0.000, C 0.000 }
gfCNCPoint1[15190] = {X 521.5668, Y 24.5714, Z -1.3333, A 0.000, B 0.000, C 0.000 }
gfCNCPoint1[15191] = {X 521.6739, Y 23.6153, Z -1.3333, A 0.000, B 0.000, C 0.000 }
gfCNCPoint1[15192] = {X 521.9900, Y 22.7066, Z -1.3333, A 0.000, B 0.000, C 0.000 }
gfCNCPoint1[15193] = {X 522.4994, Y 21.8904, Z -1.3333, A 0.000, B 0.000, C 0.000 }
gfCNCPoint1[15194] = {X 523.1768, Y 21.2071, Z -1.3333, A 0.000, B 0.000, C 0.000 }
gfCNCPoint1[15195] = {X 523.9886, Y 20.6908, Z -1.3333, A 0.000, B 0.000, C 0.000 }
gfCNCPoint1[15196] = {X 524.8946, Y 20.3669, Z -1.3333, A 0.000, B 0.000, C 0.000 }
gfCNCPoint1[15197] = {X 525.8498, Y 20.2516, Z -1.3333, A 0.000, B 0.000, C 0.000 }
gfCNCPoint1[15198] = {X 526.5695, Y 20.2516, Z -1.3333, A 0.000, B 0.000, C 0.000 }
gfCNCPoint1[15199] = {X 527.3948, Y 20.3392, Z -1.3333, A 0.000, B 0.000, C 0.000 }
gfCNCPoint1[15200] = {X 528.1881, Y 20.5830, Z -1.3333, A 0.000, B 0.000, C 0.000 }
gfCNCPoint1[15201] = {X 528.9202, Y 20.9740, Z -1.3333, A 0.000, B 0.000, C 0.000 }
gfCNCPoint1[15202] = {X 529.5640, Y 21.4978, Z -1.3333, A 0.000, B 0.000, C 0.000 }
gfCNCPoint1[15203] = {X 530.0958, Y 22.1350, Z -1.3333, A 0.000, B 0.000, C 0.000 }
gfCNCPoint1[15204] = {X 534.6319, Y 22.1354, Z -1.3333, A 0.000, B 0.000, C 0.000 }
gfCNCPoint1[15205] = {X 534.6319, Y 19.7009, Z -1.3333, A 0.000, B 0.000, C 0.000 }
gfCNCPoint1[15206] = {X 524.1929, Y 19.7004, Z -1.3333, A 0.000, B 0.000, C 0.000 }
gfCNCPoint1[15207] = {X 523.6605, Y 20.3454, Z -1.3333, A 0.000, B 0.000, C 0.000 }
gfCNCPoint1[15208] = {X 523.0138, Y 20.8757, Z -1.3333, A 0.000, B 0.000, C 0.000 }
gfCNCPoint1[15209] = {X 522.2770, Y 21.2715, Z -1.3333, A 0.000, B 0.000, C 0.000 }
gfCNCPoint1[15210] = {X 521.4777, Y 21.5178, Z -1.3333, A 0.000, B 0.000, C 0.000 }
gfCNCPoint1[15211] = {X 520.6460, Y 21.6056, Z -1.3333, A 0.000, B 0.000, C 0.000 }
gfCNCPoint1[15212] = {X 519.9691, Y 21.6057, Z -1.3333, A 0.000, B 0.000, C 0.000 }
gfCNCPoint1[15213] = {X 519.0078, Y 21.4974, Z -1.3333, A 0.000, B 0.000, C 0.000 }
gfCNCPoint1[15214] = {X 518.0947, Y 21.1779, Z -1.3333, A 0.000, B 0.000, C 0.000 }
gfCNCPoint1[15215] = {X 517.2756, Y 20.6632, Z -1.3333, A 0.000, B 0.000, C 0.000 }
gfCNCPoint1[15216] = {X 516.5916, Y 19.9792, Z -1.3333, A 0.000, B 0.000, C 0.000 }
gfCNCPoint1[15217] = {X 516.0769, Y 19.1601, Z -1.3333, A 0.000, B 0.000, C 0.000 }
gfCNCPoint1[15218] = {X 515.7574, Y 18.2470, Z -1.3333, A 0.000, B 0.000, C 0.000 }
gfCNCPoint1[15219] = {X 515.6491, Y 17.2857, Z -1.3333, A 0.000, B 0.000, C 0.000 }
gfCNCPoint1[15220] = {X 515.6491, Y 10.3077, Z -1.3333, A 0.000, B 0.000, C 0.000 }
gfCNCPoint1[15221] = {X 515.7562, Y 9.3519, Z -1.3333, A 0.000, B 0.000, C 0.000 }
gfCNCPoint1[15222] = {X 516.0720, Y 8.4435, Z -1.3333, A 0.000, B 0.000, C 0.000 }
gfCNCPoint1[15223] = {X 516.5811, Y 7.6275, Z -1.3333, A 0.000, B 0.000, C 0.000 }
gfCNCPoint1[15224] = {X 517.2580, Y 6.9443, Z -1.3333, A 0.000, B 0.000, C 0.000 }
gfCNCPoint1[15225] = {X 518.0693, Y 6.4278, Z -1.3333, A 0.000, B 0.000, C 0.000 }
gfCNCPoint1[15226] = {X 518.9748, Y 6.1037, Z -1.3333, A 0.000, B 0.000, C 0.000 }
gfCNCPoint1[15227] = {X 519.9296, Y 5.9879, Z -1.3333, A 0.000, B 0.000, C 0.000 }
gfCNCPoint1[15228] = {X 520.6502, Y 5.9879, Z -1.3333, A 0.000, B 0.000, C 0.000 }
gfCNCPoint1[15229] = {X 521.4759, Y 6.0752, Z -1.3333, A 0.000, B 0.000, C 0.000 }
gfCNCPoint1[15230] = {X 522.2696, Y 6.3189, Z -1.3333, A 0.000, B 0.000, C 0.000 }
gfCNCPoint1[15231] = {X 523.0021, Y 6.7099, Z -1.3333, A 0.000, B 0.000, C 0.000 }
gfCNCPoint1[15232] = {X 523.6462, Y 7.2338, Z -1.3333, A 0.000, B 0.000, C 0.000 }
gfCNCPoint1[15233] = {X 524.1782, Y 7.8713, Z -1.3333, A 0.000, B 0.000, C 0.000 }
gfCNCPoint1[15234] = {X 533.9641, Y 7.8716, Z -1.3333, A 0.000, B 0.000, C 0.000 }
gfCNCPoint1[15235] = {X 533.9642, Y 3.8716, Z -1.3333, A 0.000, B 0.000, C 0.000 }
gfCNCPoint1[15236] = {X 533.9641, Y 7.9516, Z -1.3333, A 0.000, B 0.000, C 0.000 }
gfCNCPoint1[15237] = {X 543.7510, Y 7.9519, Z -1.3333, A 0.000, B 0.000, C 0.000 }
gfCNCPoint1[15238] = {X 544.7131, Y 8.0356, Z -1.3333, A 0.000, B 0.000, C 0.000 }
gfCNCPoint1[15239] = {X 545.6313, Y 8.3346, Z -1.3333, A 0.000, B 0.000, C 0.000 }
gfCNCPoint1[15240] = {X 546.4582, Y 8.8334, Z -1.3333, A 0.000, B 0.000, C 0.000 }
gfCNCPoint1[15241] = {X 547.1510, Y 9.5062, Z -1.3333, A 0.000, B 0.000, C 0.000 }
gfCNCPoint1[15242] = {X 547.6738, Y 10.3181, Z -1.3333, A 0.000, B 0.000, C 0.000 }
gfCNCPoint1[15243] = {X 547.9996, Y 11.2272, Z -1.3333, A 0.000, B 0.000, C 0.000 }
gfCNCPoint1[15244] = {X 548.1114, Y 12.1864, Z -1.3333, A 0.000, B 0.000, C 0.000 }
gfCNCPoint1[15245] = {X 548.1112, Y 13.0217, Z -1.3333, A 0.000, B 0.000, C 0.000 }
gfCNCPoint1[15246] = {X 548.0026, Y 13.9321, Z -1.3333, A 0.000, B 0.000, C 0.000 }
gfCNCPoint1[15247] = {X 547.7008, Y 14.7978, Z -1.3333, A 0.000, B 0.000, C 0.000 }
gfCNCPoint1[15248] = {X 547.2200, Y 15.5785, Z -1.3333, A 0.000, B 0.000, C 0.000 }
gfCNCPoint1[15249] = {X 546.5826, Y 16.2375, Z -1.3333, A 0.000, B 0.000, C 0.000 }
gfCNCPoint1[15250] = {X 546.5828, Y 40.9512, Z -1.3333, A 0.000, B 0.000, C 0.000 }
gfCNCPoint1[15251] = {X 546.6342, Y 40.9924, Z -1.3333, A 0.000, B 0.000, C 0.000 }
gfCNCPoint1[15252] = {X 547.2522, Y 41.6499, Z -1.3333, A 0.000, B 0.000, C 0.000 }
gfCNCPoint1[15253] = {X 547.7171, Y 42.4233, Z -1.3333, A 0.000, B 0.000, C 0.000 }
gfCNCPoint1[15254] = {X 548.0079, Y 43.2775, Z -1.3333, A 0.000, B 0.000, C 0.000 }
gfCNCPoint1[15255] = {X 548.1113, Y 44.1740, Z -1.3333, A 0.000, B 0.000, C 0.000 }
gfCNCPoint1[15256] = {X 548.1114, Y 45.0005, Z -1.3333, A 0.000, B 0.000, C 0.000 }
gfCNCPoint1[15257] = {X 547.9995, Y 45.9596, Z -1.3333, A 0.000, B 0.000, C 0.000 }
gfCNCPoint1[15258] = {X 547.6738, Y 46.8687, Z -1.3333, A 0.000, B 0.000, C 0.000 }
gfCNCPoint1[15259] = {X 547.1510, Y 47.6806, Z -1.3333, A 0.000, B 0.000, C 0.000 }
gfCNCPoint1[15260] = {X 546.4582, Y 48.3533, Z -1.3333, A 0.000, B 0.000, C 0.000 }
gfCNCPoint1[15261] = {X 545.6313, Y 48.8520, Z -1.3333, A 0.000, B 0.000, C 0.000 }
gfCNCPoint1[15262] = {X 544.7130, Y 49.1509, Z -1.3333, A 0.000, B 0.000, C 0.000 }
gfCNCPoint1[15263] = {X 543.7510, Y 49.2346, Z -1.3333, A 0.000, B 0.000, C 0.000 }
gfCNCPoint1[15264] = {X 524.0030, Y 49.2352, Z -1.3333, A 0.000, B 0.000, C 0.000 }
gfCNCPoint1[15265] = {X 523.4664, Y 49.8685, Z -1.3333, A 0.000, B 0.000, C 0.000 }
gfCNCPoint1[15266] = {X 522.8203, Y 50.3897, Z -1.3333, A 0.000, B 0.000, C 0.000 }
gfCNCPoint1[15267] = {X 522.0879, Y 50.7803, Z -1.3333, A 0.000, B 0.000, C 0.000 }
gfCNCPoint1[15268] = {X 521.2951, Y 51.0264, Z -1.3333, A 0.000, B 0.000, C 0.000 }
gfCNCPoint1[15269] = {X 520.4702, Y 51.1191, Z -1.3333, A 0.000, B 0.000, C 0.000 }
gfCNCPoint1[15270] = {X 519.7998, Y 51.1191, Z -1.3333, A 0.000, B 0.000, C 0.000 }
gfCNCPoint1[15271] = {X 518.8563, Y 51.0128, Z -1.3333, A 0.000, B 0.000, C 0.000 }
gfCNCPoint1[15272] = {X 517.9601, Y 50.6992, Z -1.3333, A 0.000, B 0.000, C 0.000 }
gfCNCPoint1[15273] = {X 517.1562, Y 50.1941, Z -1.3333, A 0.000, B 0.000, C 0.000 }
gfCNCPoint1[15274] = {X 516.4848, Y 49.5227, Z -1.3333, A 0.000, B 0.000, C 0.000 }
gfCNCPoint1[15275] = {X 515.9797, Y 48.7188, Z -1.3333, A 0.000, B 0.000, C 0.000 }
gfCNCPoint1[15276] = {X 515.6661, Y 47.8226, Z -1.3333, A 0.000, B 0.000, C 0.000 }
gfCNCPoint1[15277] = {X 515.5598, Y 46.8791, Z -1.3333, A 0.000, B 0.000, C 0.000 }
gfCNCPoint1[15278] = {X 515.5598, Y 39.9011, Z -1.3333, A 0.000, B 0.000, C 0.000 }
gfCNCPoint1[15279] = {X 515.6649, Y 38.9628, Z -1.3333, A 0.000, B 0.000, C 0.000 }
gfCNCPoint1[15280] = {X 515.9751, Y 38.0710, Z -1.3333, A 0.000, B 0.000, C 0.000 }
gfCNCPoint1[15281] = {X 516.4749, Y 37.2700, Z -1.3333, A 0.000, B 0.000, C 0.000 }
gfCNCPoint1[15282] = {X 517.1395, Y 36.5995, Z -1.3333, A 0.000, B 0.000, C 0.000 }
gfCNCPoint1[15283] = {X 517.9361, Y 36.0926, Z -1.3333, A 0.000, B 0.000, C 0.000 }
gfCNCPoint1[15284] = {X 518.8251, Y 35.7746, Z -1.3333, A 0.000, B 0.000, C 0.000 }
gfCNCPoint1[15285] = {X 519.7624, Y 35.6613, Z -1.3333, A 0.000, B 0.000, C 0.000 }
gfCNCPoint1[15286] = {X 520.5258, Y 35.6615, Z -1.3333, A 0.000, B 0.000, C 0.000 }
gfCNCPoint1[15287] = {X 521.3455, Y 35.7529, Z -1.3333, A 0.000, B 0.000, C 0.000 }
gfCNCPoint1[15288] = {X 522.1321, Y 36.0012, Z -1.3333, A 0.000, B 0.000, C 0.000 }
gfCNCPoint1[15289] = {X 522.8556, Y 36.3971, Z -1.3333, A 0.000, B 0.000, C 0.000 }
gfCNCPoint1[15290] = {X 523.4888, Y 36.9257, Z -1.3333, A 0.000, B 0.000, C 0.000 }
gfCNCPoint1[15291] = {X 524.0078, Y 37.5668, Z -1.3333, A 0.000, B 0.000, C 0.000 }
gfCNCPoint1[15292] = {X 534.7119, Y 37.5674, Z -1.3333, A 0.000, B 0.000, C 0.000 }
gfCNCPoint1[15293] = {X 534.7119, Y 33.8845, Z -1.3333, A 0.000, B 0.000, C 0.000 }
gfCNCPoint1[15294] = {X 530.0661, Y 33.8839, Z -1.3333, A 0.000, B 0.000, C 0.000 }
gfCNCPoint1[15295] = {X 530.0422, Y 33.9224, Z -1.3333, A 0.000, B 0.000, C 0.000 }
gfCNCPoint1[15296] = {X 529.5199, Y 34.5542, Z -1.3333, A 0.000, B 0.000, C 0.000 }
gfCNCPoint1[15297] = {X 528.8857, Y 35.0738, Z -1.3333, A 0.000, B 0.000, C 0.000 }
gfCNCPoint1[15298] = {X 528.1634, Y 35.4615, Z -1.3333, A 0.000, B 0.000, C 0.000 }
gfCNCPoint1[15299] = {X 527.3800, Y 35.7031, Z -1.3333, A 0.000, B 0.000, C 0.000 }
gfCNCPoint1[15300] = {X 526.5648, Y 35.7893, Z -1.3333, A 0.000, B 0.000, C 0.000 }
gfCNCPoint1[15301] = {X 525.8868, Y 35.7894, Z -1.3333, A 0.000, B 0.000, C 0.000 }
gfCNCPoint1[15302] = {X 524.9433, Y 35.6831, Z -1.3333, A 0.000, B 0.000, C 0.000 }
gfCNCPoint1[15303] = {X 524.0471, Y 35.3696, Z -1.3333, A 0.000, B 0.000, C 0.000 }
gfCNCPoint1[15304] = {X 523.2432, Y 34.8644, Z -1.3333, A 0.000, B 0.000, C 0.000 }
gfCNCPoint1[15305] = {X 522.5718, Y 34.1930, Z -1.3333, A 0.000, B 0.000, C 0.000 }
gfCNCPoint1[15306] = {X 522.0666, Y 33.3891, Z -1.3333, A 0.000, B 0.000, C 0.000 }
gfCNCPoint1[15307] = {X 521.7531, Y 32.4929, Z -1.3333, A 0.000, B 0.000, C 0.000 }
gfCNCPoint1[15308] = {X 521.6468, Y 31.5495, Z -1.3333, A 0.000, B 0.000, C 0.000 }
gfCNCPoint1[15309] = {X 521.6468, Y 24.5714, Z -1.3333, A 0.000, B 0.000, C 0.000 }
gfCNCPoint1[15310] = {X 521.7519, Y 23.6330, Z -1.3333, A 0.000, B 0.000, C 0.000 }
gfCNCPoint1[15311] = {X 522.0622, Y 22.7411, Z -1.3333, A 0.000, B 0.000, C 0.000 }
gfCNCPoint1[15312] = {X 522.5621, Y 21.9400, Z -1.3333, A 0.000, B 0.000, C 0.000 }
gfCNCPoint1[15313] = {X 523.2270, Y 21.2694, Z -1.3333, A 0.000, B 0.000, C 0.000 }
gfCNCPoint1[15314] = {X 524.0238, Y 20.7626, Z -1.3333, A 0.000, B 0.000, C 0.000 }
gfCNCPoint1[15315] = {X 524.9130, Y 20.4448, Z -1.3333, A 0.000, B 0.000, C 0.000 }
gfCNCPoint1[15316] = {X 525.8505, Y 20.3316, Z -1.3333, A 0.000, B 0.000, C 0.000 }
gfCNCPoint1[15317] = {X 526.5687, Y 20.3316, Z -1.3333, A 0.000, B 0.000, C 0.000 }
gfCNCPoint1[15318] = {X 527.3870, Y 20.4193, Z -1.3333, A 0.000, B 0.000, C 0.000 }
gfCNCPoint1[15319] = {X 528.1729, Y 20.6633, Z -1.3333, A 0.000, B 0.000, C 0.000 }
gfCNCPoint1[15320] = {X 528.8969, Y 21.0546, Z -1.3333, A 0.000, B 0.000, C 0.000 }
gfCNCPoint1[15321] = {X 529.5317, Y 21.5784, Z -1.3333, A 0.000, B 0.000, C 0.000 }
gfCNCPoint1[15322] = {X 530.0533, Y 22.2150, Z -1.3333, A 0.000, B 0.000, C 0.000 }
gfCNCPoint1[15323] = {X 534.7119, Y 22.2154, Z -1.3333, A 0.000, B 0.000, C 0.000 }
gfCNCPoint1[15324] = {X 534.7119, Y 19.6209, Z -1.3333, A 0.000, B 0.000, C 0.000 }
gfCNCPoint1[15325] = {X 524.1497, Y 19.6204, Z -1.3333, A 0.000, B 0.000, C 0.000 }
gfCNCPoint1[15326] = {X 524.1266, Y 19.6557, Z -1.3333, A 0.000, B 0.000, C 0.000 }
gfCNCPoint1[15327] = {X 523.6040, Y 20.2887, Z -1.3333, A 0.000, B 0.000, C 0.000 }
gfCNCPoint1[15328] = {X 522.9693, Y 20.8092, Z -1.3333, A 0.000, B 0.000, C 0.000 }
gfCNCPoint1[15329] = {X 522.2461, Y 21.1977, Z -1.3333, A 0.000, B 0.000, C 0.000 }
gfCNCPoint1[15330] = {X 521.4617, Y 21.4395, Z -1.3333, A 0.000, B 0.000, C 0.000 }
gfCNCPoint1[15331] = {X 520.6453, Y 21.5256, Z -1.3333, A 0.000, B 0.000, C 0.000 }
gfCNCPoint1[15332] = {X 519.9691, Y 21.5257, Z -1.3333, A 0.000, B 0.000, C 0.000 }
gfCNCPoint1[15333] = {X 519.0256, Y 21.4194, Z -1.3333, A 0.000, B 0.000, C 0.000 }
gfCNCPoint1[15334] = {X 518.1294, Y 21.1058, Z -1.3333, A 0.000, B 0.000, C 0.000 }
gfCNCPoint1[15335] = {X 517.3255, Y 20.6007, Z -1.3333, A 0.000, B 0.000, C 0.000 }
gfCNCPoint1[15336] = {X 516.6541, Y 19.9293, Z -1.3333, A 0.000, B 0.000, C 0.000 }
gfCNCPoint1[15337] = {X 516.1490, Y 19.1254, Z -1.3333, A 0.000, B 0.000, C 0.000 }
gfCNCPoint1[15338] = {X 515.8354, Y 18.2292, Z -1.3333, A 0.000, B 0.000, C 0.000 }
gfCNCPoint1[15339] = {X 515.7291, Y 17.2857, Z -1.3333, A 0.000, B 0.000, C 0.000 }
gfCNCPoint1[15340] = {X 515.7291, Y 10.3077, Z -1.3333, A 0.000, B 0.000, C 0.000 }
gfCNCPoint1[15341] = {X 515.8342, Y 9.3696, Z -1.3333, A 0.000, B 0.000, C 0.000 }
gfCNCPoint1[15342] = {X 516.1442, Y 8.4780, Z -1.3333, A 0.000, B 0.000, C 0.000 }
gfCNCPoint1[15343] = {X 516.6438, Y 7.6771, Z -1.3333, A 0.000, B 0.000, C 0.000 }
gfCNCPoint1[15344] = {X 517.3082, Y 7.0066, Z -1.3333, A 0.000, B 0.000, C 0.000 }
gfCNCPoint1[15345] = {X 518.1045, Y 6.4997, Z -1.3333, A 0.000, B 0.000, C 0.000 }
gfCNCPoint1[15346] = {X 518.9932, Y 6.1815, Z -1.3333, A 0.000, B 0.000, C 0.000 }
gfCNCPoint1[15347] = {X 519.9303, Y 6.0679, Z -1.3333, A 0.000, B 0.000, C 0.000 }
gfCNCPoint1[15348] = {X 520.6494, Y 6.0679, Z -1.3333, A 0.000, B 0.000, C 0.000 }
gfCNCPoint1[15349] = {X 521.4681, Y 6.1553, Z -1.3333, A 0.000, B 0.000, C 0.000 }
gfCNCPoint1[15350] = {X 522.2544, Y 6.3992, Z -1.3333, A 0.000, B 0.000, C 0.000 }
gfCNCPoint1[15351] = {X 522.9788, Y 6.7906, Z -1.3333, A 0.000, B 0.000, C 0.000 }
gfCNCPoint1[15352] = {X 523.6138, Y 7.3145, Z -1.3333, A 0.000, B 0.000, C 0.000 }
gfCNCPoint1[15353] = {X 524.1357, Y 7.9513, Z -1.3333, A 0.000, B 0.000, C 0.000 }
gfCNCPoint1[15354] = {X 533.9641, Y 7.9516, Z -1.3333, A 0.000, B 0.000, C 0.000 }
gfCNCPoint1[15355] = {X 533.9642, Y 3.9516, Z -1.3333, A 0.000, B 0.000, C 0.000 }
gfCNCPoint1[15356] = {X 533.9641, Y 8.0316, Z -1.3333, A 0.000, B 0.000, C 0.000 }
gfCNCPoint1[15357] = {X 543.7521, Y 8.0319, Z -1.3333, A 0.000, B 0.000, C 0.000 }
gfCNCPoint1[15358] = {X 544.6962, Y 8.1138, Z -1.3333, A 0.000, B 0.000, C 0.000 }
gfCNCPoint1[15359] = {X 545.5974, Y 8.4071, Z -1.3333, A 0.000, B 0.000, C 0.000 }
gfCNCPoint1[15360] = {X 546.4089, Y 8.8964, Z -1.3333, A 0.000, B 0.000, C 0.000 }
gfCNCPoint1[15361] = {X 547.0888, Y 9.5565, Z -1.3333, A 0.000, B 0.000, C 0.000 }
gfCNCPoint1[15362] = {X 547.6019, Y 10.3532, Z -1.3333, A 0.000, B 0.000, C 0.000 }
gfCNCPoint1[15363] = {X 547.9216, Y 11.2453, Z -1.3333, A 0.000, B 0.000, C 0.000 }
gfCNCPoint1[15364] = {X 548.0314, Y 12.1865, Z -1.3333, A 0.000, B 0.000, C 0.000 }
gfCNCPoint1[15365] = {X 548.0312, Y 13.0208, Z -1.3333, A 0.000, B 0.000, C 0.000 }
gfCNCPoint1[15366] = {X 547.9287, Y 13.8968, Z -1.3333, A 0.000, B 0.000, C 0.000 }
gfCNCPoint1[15367] = {X 547.6439, Y 14.7314, Z -1.3333, A 0.000, B 0.000, C 0.000 }
gfCNCPoint1[15368] = {X 547.1895, Y 15.4872, Z -1.3333, A 0.000, B 0.000, C 0.000 }
gfCNCPoint1[15369] = {X 546.5860, Y 16.1303, Z -1.3333, A 0.000, B 0.000, C 0.000 }
gfCNCPoint1[15370] = {X 546.5026, Y 16.2002, Z -1.3333, A 0.000, B 0.000, C 0.000 }
gfCNCPoint1[15371] = {X 546.5028, Y 40.9896, Z -1.3333, A 0.000, B 0.000, C 0.000 }
gfCNCPoint1[15372] = {X 546.5830, Y 41.0540, Z -1.3333, A 0.000, B 0.000, C 0.000 }
gfCNCPoint1[15373] = {X 547.1890, Y 41.6990, Z -1.3333, A 0.000, B 0.000, C 0.000 }
gfCNCPoint1[15374] = {X 547.6449, Y 42.4576, Z -1.3333, A 0.000, B 0.000, C 0.000 }
gfCNCPoint1[15375] = {X 547.9299, Y 43.2954, Z -1.3333, A 0.000, B 0.000, C 0.000 }
gfCNCPoint1[15376] = {X 548.0313, Y 44.1746, Z -1.3333, A 0.000, B 0.000, C 0.000 }
gfCNCPoint1[15377] = {X 548.0314, Y 45.0003, Z -1.3333, A 0.000, B 0.000, C 0.000 }
gfCNCPoint1[15378] = {X 547.9216, Y 45.9415, Z -1.3333, A 0.000, B 0.000, C 0.000 }
gfCNCPoint1[15379] = {X 547.6019, Y 46.8336, Z -1.3333, A 0.000, B 0.000, C 0.000 }
gfCNCPoint1[15380] = {X 547.0888, Y 47.6302, Z -1.3333, A 0.000, B 0.000, C 0.000 }
gfCNCPoint1[15381] = {X 546.4088, Y 48.2903, Z -1.3333, A 0.000, B 0.000, C 0.000 }
gfCNCPoint1[15382] = {X 545.5973, Y 48.7796, Z -1.3333, A 0.000, B 0.000, C 0.000 }
gfCNCPoint1[15383] = {X 544.6962, Y 49.0727, Z -1.3333, A 0.000, B 0.000, C 0.000 }
gfCNCPoint1[15384] = {X 543.7521, Y 49.1546, Z -1.3333, A 0.000, B 0.000, C 0.000 }
gfCNCPoint1[15385] = {X 523.9610, Y 49.1552, Z -1.3333, A 0.000, B 0.000, C 0.000 }
gfCNCPoint1[15386] = {X 523.4343, Y 49.7878, Z -1.3333, A 0.000, B 0.000, C 0.000 }
gfCNCPoint1[15387] = {X 522.7972, Y 50.3090, Z -1.3333, A 0.000, B 0.000, C 0.000 }
gfCNCPoint1[15388] = {X 522.0728, Y 50.6999, Z -1.3333, A 0.000, B 0.000, C 0.000 }
gfCNCPoint1[15389] = {X 521.2874, Y 50.9462, Z -1.3333, A 0.000, B 0.000, C 0.000 }
gfCNCPoint1[15390] = {X 520.4695, Y 51.0391, Z -1.3333, A 0.000, B 0.000, C 0.000 }
gfCNCPoint1[15391] = {X 519.7998, Y 51.0391, Z -1.3333, A 0.000, B 0.000, C 0.000 }
gfCNCPoint1[15392] = {X 518.8741, Y 50.9348, Z -1.3333, A 0.000, B 0.000, C 0.000 }
gfCNCPoint1[15393] = {X 517.9948, Y 50.6272, Z -1.3333, A 0.000, B 0.000, C 0.000 }
gfCNCPoint1[15394] = {X 517.2061, Y 50.1315, Z -1.3333, A 0.000, B 0.000, C 0.000 }
gfCNCPoint1[15395] = {X 516.5474, Y 49.4728, Z -1.3333, A 0.000, B 0.000, C 0.000 }
gfCNCPoint1[15396] = {X 516.0517, Y 48.6841, Z -1.3333, A 0.000, B 0.000, C 0.000 }
gfCNCPoint1[15397] = {X 515.7441, Y 47.8048, Z -1.3333, A 0.000, B 0.000, C 0.000 }
gfCNCPoint1[15398] = {X 515.6398, Y 46.8791, Z -1.3333, A 0.000, B 0.000, C 0.000 }
gfCNCPoint1[15399] = {X 515.6398, Y 39.9011, Z -1.3333, A 0.000, B 0.000, C 0.000 }
gfCNCPoint1[15400] = {X 515.7429, Y 38.9805, Z -1.3333, A 0.000, B 0.000, C 0.000 }
gfCNCPoint1[15401] = {X 516.0472, Y 38.1056, Z -1.3333, A 0.000, B 0.000, C 0.000 }
gfCNCPoint1[15402] = {X 516.5376, Y 37.3197, Z -1.3333, A 0.000, B 0.000, C 0.000 }
gfCNCPoint1[15403] = {X 517.1897, Y 36.6618, Z -1.3333, A 0.000, B 0.000, C 0.000 }
gfCNCPoint1[15404] = {X 517.9713, Y 36.1645, Z -1.3333, A 0.000, B 0.000, C 0.000 }
gfCNCPoint1[15405] = {X 518.8435, Y 35.8525, Z -1.3333, A 0.000, B 0.000, C 0.000 }
gfCNCPoint1[15406] = {X 519.7631, Y 35.7413, Z -1.3333, A 0.000, B 0.000, C 0.000 }
gfCNCPoint1[15407] = {X 520.5247, Y 35.7415, Z -1.3333, A 0.000, B 0.000, C 0.000 }
gfCNCPoint1[15408] = {X 521.3374, Y 35.8329, Z -1.3333, A 0.000, B 0.000, C 0.000 }
gfCNCPoint1[15409] = {X 522.1164, Y 36.0816, Z -1.3333, A 0.000, B 0.000, C 0.000 }
gfCNCPoint1[15410] = {X 522.8318, Y 36.4778, Z -1.3333, A 0.000, B 0.000, C 0.000 }
gfCNCPoint1[15411] = {X 523.4558, Y 37.0064, Z -1.3333, A 0.000, B 0.000, C 0.000 }
gfCNCPoint1[15412] = {X 523.9644, Y 37.6468, Z -1.3333, A 0.000, B 0.000, C 0.000 }
gfCNCPoint1[15413] = {X 534.7919, Y 37.6474, Z -1.3333, A 0.000, B 0.000, C 0.000 }
gfCNCPoint1[15414] = {X 534.7919, Y 33.8045, Z -1.3333, A 0.000, B 0.000, C 0.000 }
gfCNCPoint1[15415] = {X 530.0216, Y 33.8039, Z -1.3333, A 0.000, B 0.000, C 0.000 }
gfCNCPoint1[15416] = {X 529.9751, Y 33.8789, Z -1.3333, A 0.000, B 0.000, C 0.000 }
gfCNCPoint1[15417] = {X 529.4626, Y 34.4984, Z -1.3333, A 0.000, B 0.000, C 0.000 }
gfCNCPoint1[15418] = {X 528.8405, Y 35.0078, Z -1.3333, A 0.000, B 0.000, C 0.000 }
gfCNCPoint1[15419] = {X 528.1320, Y 35.3879, Z -1.3333, A 0.000, B 0.000, C 0.000 }
gfCNCPoint1[15420] = {X 527.3637, Y 35.6247, Z -1.3333, A 0.000, B 0.000, C 0.000 }
gfCNCPoint1[15421] = {X 526.5641, Y 35.7093, Z -1.3333, A 0.000, B 0.000, C 0.000 }
gfCNCPoint1[15422] = {X 525.8868, Y 35.7094, Z -1.3333, A 0.000, B 0.000, C 0.000 }
gfCNCPoint1[15423] = {X 524.9611, Y 35.6051, Z -1.3333, A 0.000, B 0.000, C 0.000 }
gfCNCPoint1[15424] = {X 524.0818, Y 35.2975, Z -1.3333, A 0.000, B 0.000, C 0.000 }
gfCNCPoint1[15425] = {X 523.2930, Y 34.8019, Z -1.3333, A 0.000, B 0.000, C 0.000 }
gfCNCPoint1[15426] = {X 522.6343, Y 34.1432, Z -1.3333, A 0.000, B 0.000, C 0.000 }
gfCNCPoint1[15427] = {X 522.1387, Y 33.3544, Z -1.3333, A 0.000, B 0.000, C 0.000 }
gfCNCPoint1[15428] = {X 521.8311, Y 32.4751, Z -1.3333, A 0.000, B 0.000, C 0.000 }
gfCNCPoint1[15429] = {X 521.7268, Y 31.5495, Z -1.3333, A 0.000, B 0.000, C 0.000 }
gfCNCPoint1[15430] = {X 521.7268, Y 24.5714, Z -1.3333, A 0.000, B 0.000, C 0.000 }
gfCNCPoint1[15431] = {X 521.8299, Y 23.6507, Z -1.3333, A 0.000, B 0.000, C 0.000 }
gfCNCPoint1[15432] = {X 522.1343, Y 22.7756, Z -1.3333, A 0.000, B 0.000, C 0.000 }
gfCNCPoint1[15433] = {X 522.6248, Y 21.9897, Z -1.3333, A 0.000, B 0.000, C 0.000 }
gfCNCPoint1[15434] = {X 523.2772, Y 21.3317, Z -1.3333, A 0.000, B 0.000, C 0.000 }
gfCNCPoint1[15435] = {X 524.0589, Y 20.8345, Z -1.3333, A 0.000, B 0.000, C 0.000 }
gfCNCPoint1[15436] = {X 524.9313, Y 20.5226, Z -1.3333, A 0.000, B 0.000, C 0.000 }
gfCNCPoint1[15437] = {X 525.8511, Y 20.4116, Z -1.3333, A 0.000, B 0.000, C 0.000 }
gfCNCPoint1[15438] = {X 526.5679, Y 20.4116, Z -1.3333, A 0.000, B 0.000, C 0.000 }
gfCNCPoint1[15439] = {X 527.3791, Y 20.4993, Z -1.3333, A 0.000, B 0.000, C 0.000 }
gfCNCPoint1[15440] = {X 528.1576, Y 20.7437, Z -1.3333, A 0.000, B 0.000, C 0.000 }
gfCNCPoint1[15441] = {X 528.8734, Y 21.1353, Z -1.3333, A 0.000, B 0.000, C 0.000 }
gfCNCPoint1[15442] = {X 529.4990, Y 21.6591, Z -1.3333, A 0.000, B 0.000, C 0.000 }
gfCNCPoint1[15443] = {X 530.0103, Y 22.2950, Z -1.3333, A 0.000, B 0.000, C 0.000 }
gfCNCPoint1[15444] = {X 534.7919, Y 22.2954, Z -1.3333, A 0.000, B 0.000, C 0.000 }
gfCNCPoint1[15445] = {X 534.7919, Y 19.5409, Z -1.3333, A 0.000, B 0.000, C 0.000 }
gfCNCPoint1[15446] = {X 524.1052, Y 19.5404, Z -1.3333, A 0.000, B 0.000, C 0.000 }
gfCNCPoint1[15447] = {X 524.0767, Y 19.5864, Z -1.3333, A 0.000, B 0.000, C 0.000 }
gfCNCPoint1[15448] = {X 523.5643, Y 20.2153, Z -1.3333, A 0.000, B 0.000, C 0.000 }
gfCNCPoint1[15449] = {X 522.9395, Y 20.7328, Z -1.3333, A 0.000, B 0.000, C 0.000 }
gfCNCPoint1[15450] = {X 522.2262, Y 21.1193, Z -1.3333, A 0.000, B 0.000, C 0.000 }
gfCNCPoint1[15451] = {X 521.4514, Y 21.3599, Z -1.3333, A 0.000, B 0.000, C 0.000 }
gfCNCPoint1[15452] = {X 520.6447, Y 21.4456, Z -1.3333, A 0.000, B 0.000, C 0.000 }
gfCNCPoint1[15453] = {X 519.9691, Y 21.4457, Z -1.3333, A 0.000, B 0.000, C 0.000 }
gfCNCPoint1[15454] = {X 519.0434, Y 21.3414, Z -1.3333, A 0.000, B 0.000, C 0.000 }
gfCNCPoint1[15455] = {X 518.1641, Y 21.0337, Z -1.3333, A 0.000, B 0.000, C 0.000 }
gfCNCPoint1[15456] = {X 517.3754, Y 20.5381, Z -1.3333, A 0.000, B 0.000, C 0.000 }
gfCNCPoint1[15457] = {X 516.7167, Y 19.8794, Z -1.3333, A 0.000, B 0.000, C 0.000 }
gfCNCPoint1[15458] = {X 516.2211, Y 19.0907, Z -1.3333, A 0.000, B 0.000, C 0.000 }
gfCNCPoint1[15459] = {X 515.9134, Y 18.2114, Z -1.3333, A 0.000, B 0.000, C 0.000 }
gfCNCPoint1[15460] = {X 515.8091, Y 17.2857, Z -1.3333, A 0.000, B 0.000, C 0.000 }
gfCNCPoint1[15461] = {X 515.8091, Y 10.3077, Z -1.3333, A 0.000, B 0.000, C 0.000 }
gfCNCPoint1[15462] = {X 515.9122, Y 9.3873, Z -1.3333, A 0.000, B 0.000, C 0.000 }
gfCNCPoint1[15463] = {X 516.2164, Y 8.5125, Z -1.3333, A 0.000, B 0.000, C 0.000 }
gfCNCPoint1[15464] = {X 516.7065, Y 7.7267, Z -1.3333, A 0.000, B 0.000, C 0.000 }
gfCNCPoint1[15465] = {X 517.3584, Y 7.0689, Z -1.3333, A 0.000, B 0.000, C 0.000 }
gfCNCPoint1[15466] = {X 518.1397, Y 6.5715, Z -1.3333, A 0.000, B 0.000, C 0.000 }
gfCNCPoint1[15467] = {X 519.0117, Y 6.2594, Z -1.3333, A 0.000, B 0.000, C 0.000 }
gfCNCPoint1[15468] = {X 519.9311, Y 6.1479, Z -1.3333, A 0.000, B 0.000, C 0.000 }
gfCNCPoint1[15469] = {X 520.6487, Y 6.1479, Z -1.3333, A 0.000, B 0.000, C 0.000 }
gfCNCPoint1[15470] = {X 521.4603, Y 6.2353, Z -1.3333, A 0.000, B 0.000, C 0.000 }
gfCNCPoint1[15471] = {X 522.2391, Y 6.4796, Z -1.3333, A 0.000, B 0.000, C 0.000 }
gfCNCPoint1[15472] = {X 522.9553, Y 6.8713, Z -1.3333, A 0.000, B 0.000, C 0.000 }
gfCNCPoint1[15473] = {X 523.5811, Y 7.3952, Z -1.3333, A 0.000, B 0.000, C 0.000 }
gfCNCPoint1[15474] = {X 524.0927, Y 8.0313, Z -1.3333, A 0.000, B 0.000, C 0.000 }
gfCNCPoint1[15475] = {X 533.9641, Y 8.0316, Z -1.3333, A 0.000, B 0.000, C 0.000 }
gfCNCPoint1[15476] = {X 533.9642, Y 4.0316, Z -1.3333, A 0.000, B 0.000, C 0.000 }
gfCNCPoint1[15477] = {X 533.9641, Y 8.1116, Z -1.3333, A 0.000, B 0.000, C 0.000 }
gfCNCPoint1[15478] = {X 543.7532, Y 8.1119, Z -1.3333, A 0.000, B 0.000, C 0.000 }
gfCNCPoint1[15479] = {X 544.6794, Y 8.1920, Z -1.3333, A 0.000, B 0.000, C 0.000 }
gfCNCPoint1[15480] = {X 545.5634, Y 8.4795, Z -1.3333, A 0.000, B 0.000, C 0.000 }
gfCNCPoint1[15481] = {X 546.3596, Y 8.9594, Z -1.3333, A 0.000, B 0.000, C 0.000 }
gfCNCPoint1[15482] = {X 547.0266, Y 9.6068, Z -1.3333, A 0.000, B 0.000, C 0.000 }
gfCNCPoint1[15483] = {X 547.5300, Y 10.3883, Z -1.3333, A 0.000, B 0.000, C 0.000 }
gfCNCPoint1[15484] = {X 547.8437, Y 11.2634, Z -1.3333, A 0.000, B 0.000, C 0.000 }
gfCNCPoint1[15485] = {X 547.9514, Y 12.1867, Z -1.3333, A 0.000, B 0.000, C 0.000 }
gfCNCPoint1[15486] = {X 547.9512, Y 13.0200, Z -1.3333, A 0.000, B 0.000, C 0.000 }
gfCNCPoint1[15487] = {X 547.8507, Y 13.8791, Z -1.3333, A 0.000, B 0.000, C 0.000 }
gfCNCPoint1[15488] = {X 547.5713, Y 14.6977, Z -1.3333, A 0.000, B 0.000, C 0.000 }
gfCNCPoint1[15489] = {X 547.1257, Y 15.4390, Z -1.3333, A 0.000, B 0.000, C 0.000 }
gfCNCPoint1[15490] = {X 546.5338, Y 16.0697, Z -1.3333, A 0.000, B 0.000, C 0.000 }
gfCNCPoint1[15491] = {X 546.4793, Y 16.1157, Z -1.3333, A 0.000, B 0.000, C 0.000 }
gfCNCPoint1[15492] = {X 546.4241, Y 16.1609, Z -1.3333, A 0.000, B 0.000, C 0.000 }
gfCNCPoint1[15493] = {X 546.4228, Y 41.0280, Z -1.3333, A 0.000, B 0.000, C 0.000 }
gfCNCPoint1[15494] = {X 546.5319, Y 41.1155, Z -1.3333, A 0.000, B 0.000, C 0.000 }
gfCNCPoint1[15495] = {X 547.1258, Y 41.7480, Z -1.3333, A 0.000, B 0.000, C 0.000 }
gfCNCPoint1[15496] = {X 547.5726, Y 42.4919, Z -1.3333, A 0.000, B 0.000, C 0.000 }
gfCNCPoint1[15497] = {X 547.8519, Y 43.3133, Z -1.3333, A 0.000, B 0.000, C 0.000 }
gfCNCPoint1[15498] = {X 547.9513, Y 44.1753, Z -1.3333, A 0.000, B 0.000, C 0.000 }
gfCNCPoint1[15499] = {X 547.9514, Y 45.0001, Z -1.3333, A 0.000, B 0.000, C 0.000 }
gfCNCPoint1[15500] = {X 547.8437, Y 45.9234, Z -1.3333, A 0.000, B 0.000, C 0.000 }
gfCNCPoint1[15501] = {X 547.5300, Y 46.7984, Z -1.3333, A 0.000, B 0.000, C 0.000 }
gfCNCPoint1[15502] = {X 547.0266, Y 47.5799, Z -1.3333, A 0.000, B 0.000, C 0.000 }
gfCNCPoint1[15503] = {X 546.3595, Y 48.2273, Z -1.3333, A 0.000, B 0.000, C 0.000 }
gfCNCPoint1[15504] = {X 545.5634, Y 48.7071, Z -1.3333, A 0.000, B 0.000, C 0.000 }
gfCNCPoint1[15505] = {X 544.6793, Y 48.9945, Z -1.3333, A 0.000, B 0.000, C 0.000 }
gfCNCPoint1[15506] = {X 543.7532, Y 49.0746, Z -1.3333, A 0.000, B 0.000, C 0.000 }
gfCNCPoint1[15507] = {X 523.9185, Y 49.0752, Z -1.3333, A 0.000, B 0.000, C 0.000 }
gfCNCPoint1[15508] = {X 523.4020, Y 49.7070, Z -1.3333, A 0.000, B 0.000, C 0.000 }
gfCNCPoint1[15509] = {X 522.7739, Y 50.2282, Z -1.3333, A 0.000, B 0.000, C 0.000 }
gfCNCPoint1[15510] = {X 522.0576, Y 50.6194, Z -1.3333, A 0.000, B 0.000, C 0.000 }
gfCNCPoint1[15511] = {X 521.2796, Y 50.8661, Z -1.3333, A 0.000, B 0.000, C 0.000 }
gfCNCPoint1[15512] = {X 520.4688, Y 50.9591, Z -1.3333, A 0.000, B 0.000, C 0.000 }
gfCNCPoint1[15513] = {X 519.7998, Y 50.9591, Z -1.3333, A 0.000, B 0.000, C 0.000 }
gfCNCPoint1[15514] = {X 518.8919, Y 50.8568, Z -1.3333, A 0.000, B 0.000, C 0.000 }
gfCNCPoint1[15515] = {X 518.0295, Y 50.5551, Z -1.3333, A 0.000, B 0.000, C 0.000 }
gfCNCPoint1[15516] = {X 517.2559, Y 50.0690, Z -1.3333, A 0.000, B 0.000, C 0.000 }
gfCNCPoint1[15517] = {X 516.6099, Y 49.4230, Z -1.3333, A 0.000, B 0.000, C 0.000 }
gfCNCPoint1[15518] = {X 516.1238, Y 48.6494, Z -1.3333, A 0.000, B 0.000, C 0.000 }
gfCNCPoint1[15519] = {X 515.8221, Y 47.7870, Z -1.3333, A 0.000, B 0.000, C 0.000 }
gfCNCPoint1[15520] = {X 515.7198, Y 46.8791, Z -1.3333, A 0.000, B 0.000, C 0.000 }
gfCNCPoint1[15521] = {X 515.7198, Y 39.9011, Z -1.3333, A 0.000, B 0.000, C 0.000 }
gfCNCPoint1[15522] = {X 515.8209, Y 38.9982, Z -1.3333, A 0.000, B 0.000, C 0.000 }
gfCNCPoint1[15523] = {X 516.1194, Y 38.1401, Z -1.3333, A 0.000, B 0.000, C 0.000 }
gfCNCPoint1[15524] = {X 516.6003, Y 37.3693, Z -1.3333, A 0.000, B 0.000, C 0.000 }
gfCNCPoint1[15525] = {X 517.2399, Y 36.7241, Z -1.3333, A 0.000, B 0.000, C 0.000 }
gfCNCPoint1[15526] = {X 518.0064, Y 36.2364, Z -1.3333, A 0.000, B 0.000, C 0.000 }
gfCNCPoint1[15527] = {X 518.8619, Y 35.9304, Z -1.3333, A 0.000, B 0.000, C 0.000 }
gfCNCPoint1[15528] = {X 519.7638, Y 35.8213, Z -1.3333, A 0.000, B 0.000, C 0.000 }
gfCNCPoint1[15529] = {X 520.5236, Y 35.8215, Z -1.3333, A 0.000, B 0.000, C 0.000 }
gfCNCPoint1[15530] = {X 521.3291, Y 35.9130, Z -1.3333, A 0.000, B 0.000, C 0.000 }
gfCNCPoint1[15531] = {X 522.1007, Y 36.1619, Z -1.3333, A 0.000, B 0.000, C 0.000 }
gfCNCPoint1[15532] = {X 522.8078, Y 36.5585, Z -1.3333, A 0.000, B 0.000, C 0.000 }
gfCNCPoint1[15533] = {X 523.4225, Y 37.0871, Z -1.3333, A 0.000, B 0.000, C 0.000 }
gfCNCPoint1[15534] = {X 523.9205, Y 37.7268, Z -1.3333, A 0.000, B 0.000, C 0.000 }
gfCNCPoint1[15535] = {X 534.8719, Y 37.7274, Z -1.3333, A 0.000, B 0.000, C 0.000 }
gfCNCPoint1[15536] = {X 534.8719, Y 33.7245, Z -1.3333, A 0.000, B 0.000, C 0.000 }
gfCNCPoint1[15537] = {X 529.9772, Y 33.7239, Z -1.3333, A 0.000, B 0.000, C 0.000 }
gfCNCPoint1[15538] = {X 529.9071, Y 33.8366, Z -1.3333, A 0.000, B 0.000, C 0.000 }
gfCNCPoint1[15539] = {X 529.2612, Y 34.5790, Z -1.3333, A 0.000, B 0.000, C 0.000 }
gfCNCPoint1[15540] = {X 528.4563, Y 35.1452, Z -1.3333, A 0.000, B 0.000, C 0.000 }
gfCNCPoint1[15541] = {X 527.5392, Y 35.5023, Z -1.3333, A 0.000, B 0.000, C 0.000 }
gfCNCPoint1[15542] = {X 526.5634, Y 35.6293, Z -1.3333, A 0.000, B 0.000, C 0.000 }
gfCNCPoint1[15543] = {X 525.8868, Y 35.6295, Z -1.3333, A 0.000, B 0.000, C 0.000 }
gfCNCPoint1[15544] = {X 524.9789, Y 35.5272, Z -1.3333, A 0.000, B 0.000, C 0.000 }
gfCNCPoint1[15545] = {X 524.1165, Y 35.2254, Z -1.3333, A 0.000, B 0.000, C 0.000 }
gfCNCPoint1[15546] = {X 523.3429, Y 34.7393, Z -1.3333, A 0.000, B 0.000, C 0.000 }
gfCNCPoint1[15547] = {X 522.6969, Y 34.0933, Z -1.3333, A 0.000, B 0.000, C 0.000 }
gfCNCPoint1[15548] = {X 522.2108, Y 33.3197, Z -1.3333, A 0.000, B 0.000, C 0.000 }
gfCNCPoint1[15549] = {X 521.9091, Y 32.4573, Z -1.3333, A 0.000, B 0.000, C 0.000 }
gfCNCPoint1[15550] = {X 521.8068, Y 31.5495, Z -1.3333, A 0.000, B 0.000, C 0.000 }
gfCNCPoint1[15551] = {X 521.8068, Y 24.5714, Z -1.3333, A 0.000, B 0.000, C 0.000 }
gfCNCPoint1[15552] = {X 521.9079, Y 23.6684, Z -1.3333, A 0.000, B 0.000, C 0.000 }
gfCNCPoint1[15553] = {X 522.2065, Y 22.8102, Z -1.3333, A 0.000, B 0.000, C 0.000 }
gfCNCPoint1[15554] = {X 522.6876, Y 22.0393, Z -1.3333, A 0.000, B 0.000, C 0.000 }
gfCNCPoint1[15555] = {X 523.3273, Y 21.3940, Z -1.3333, A 0.000, B 0.000, C 0.000 }
gfCNCPoint1[15556] = {X 524.0941, Y 20.9064, Z -1.3333, A 0.000, B 0.000, C 0.000 }
gfCNCPoint1[15557] = {X 524.9497, Y 20.6005, Z -1.3333, A 0.000, B 0.000, C 0.000 }
gfCNCPoint1[15558] = {X 525.8518, Y 20.4916, Z -1.3333, A 0.000, B 0.000, C 0.000 }
gfCNCPoint1[15559] = {X 526.5672, Y 20.4916, Z -1.3333, A 0.000, B 0.000, C 0.000 }
gfCNCPoint1[15560] = {X 527.3712, Y 20.5794, Z -1.3333, A 0.000, B 0.000, C 0.000 }
gfCNCPoint1[15561] = {X 528.1421, Y 20.8241, Z -1.3333, A 0.000, B 0.000, C 0.000 }
gfCNCPoint1[15562] = {X 528.8496, Y 21.2161, Z -1.3333, A 0.000, B 0.000, C 0.000 }
gfCNCPoint1[15563] = {X 529.4659, Y 21.7399, Z -1.3333, A 0.000, B 0.000, C 0.000 }
gfCNCPoint1[15564] = {X 529.9667, Y 22.3750, Z -1.3333, A 0.000, B 0.000, C 0.000 }
gfCNCPoint1[15565] = {X 534.8719, Y 22.3754, Z -1.3333, A 0.000, B 0.000, C 0.000 }
gfCNCPoint1[15566] = {X 534.8719, Y 19.4610, Z -1.3333, A 0.000, B 0.000, C 0.000 }
gfCNCPoint1[15567] = {X 524.0607, Y 19.4604, Z -1.3333, A 0.000, B 0.000, C 0.000 }
gfCNCPoint1[15568] = {X 524.0087, Y 19.5442, Z -1.3333, A 0.000, B 0.000, C 0.000 }
gfCNCPoint1[15569] = {X 523.5061, Y 20.1604, Z -1.3333, A 0.000, B 0.000, C 0.000 }
gfCNCPoint1[15570] = {X 522.8935, Y 20.6674, Z -1.3333, A 0.000, B 0.000, C 0.000 }
gfCNCPoint1[15571] = {X 522.1942, Y 21.0459, Z -1.3333, A 0.000, B 0.000, C 0.000 }
gfCNCPoint1[15572] = {X 521.4348, Y 21.2816, Z -1.3333, A 0.000, B 0.000, C 0.000 }
gfCNCPoint1[15573] = {X 520.6440, Y 21.3656, Z -1.3333, A 0.000, B 0.000, C 0.000 }
gfCNCPoint1[15574] = {X 519.9691, Y 21.3657, Z -1.3333, A 0.000, B 0.000, C 0.000 }
gfCNCPoint1[15575] = {X 519.0612, Y 21.2634, Z -1.3333, A 0.000, B 0.000, C 0.000 }
gfCNCPoint1[15576] = {X 518.1989, Y 20.9617, Z -1.3333, A 0.000, B 0.000, C 0.000 }
gfCNCPoint1[15577] = {X 517.4253, Y 20.4756, Z -1.3333, A 0.000, B 0.000, C 0.000 }
gfCNCPoint1[15578] = {X 516.7792, Y 19.8296, Z -1.3333, A 0.000, B 0.000, C 0.000 }
gfCNCPoint1[15579] = {X 516.2932, Y 19.0560, Z -1.3333, A 0.000, B 0.000, C 0.000 }
gfCNCPoint1[15580] = {X 515.9914, Y 18.1936, Z -1.3333, A 0.000, B 0.000, C 0.000 }
gfCNCPoint1[15581] = {X 515.8891, Y 17.2857, Z -1.3333, A 0.000, B 0.000, C 0.000 }
gfCNCPoint1[15582] = {X 515.8891, Y 10.3077, Z -1.3333, A 0.000, B 0.000, C 0.000 }
gfCNCPoint1[15583] = {X 515.9902, Y 9.4050, Z -1.3333, A 0.000, B 0.000, C 0.000 }
gfCNCPoint1[15584] = {X 516.2885, Y 8.5471, Z -1.3333, A 0.000, B 0.000, C 0.000 }
gfCNCPoint1[15585] = {X 516.7693, Y 7.7764, Z -1.3333, A 0.000, B 0.000, C 0.000 }
gfCNCPoint1[15586] = {X 517.4086, Y 7.1312, Z -1.3333, A 0.000, B 0.000, C 0.000 }
gfCNCPoint1[15587] = {X 518.1749, Y 6.6434, Z -1.3333, A 0.000, B 0.000, C 0.000 }
gfCNCPoint1[15588] = {X 519.0301, Y 6.3372, Z -1.3333, A 0.000, B 0.000, C 0.000 }
gfCNCPoint1[15589] = {X 519.9318, Y 6.2279, Z -1.3333, A 0.000, B 0.000, C 0.000 }
gfCNCPoint1[15590] = {X 520.6480, Y 6.2279, Z -1.3333, A 0.000, B 0.000, C 0.000 }
gfCNCPoint1[15591] = {X 521.4524, Y 6.3154, Z -1.3333, A 0.000, B 0.000, C 0.000 }
gfCNCPoint1[15592] = {X 522.2236, Y 6.5600, Z -1.3333, A 0.000, B 0.000, C 0.000 }
gfCNCPoint1[15593] = {X 522.9315, Y 6.9520, Z -1.3333, A 0.000, B 0.000, C 0.000 }
gfCNCPoint1[15594] = {X 523.5481, Y 7.4760, Z -1.3333, A 0.000, B 0.000, C 0.000 }
gfCNCPoint1[15595] = {X 524.0491, Y 8.1113, Z -1.3333, A 0.000, B 0.000, C 0.000 }
gfCNCPoint1[15596] = {X 533.9641, Y 8.1116, Z -1.3333, A 0.000, B 0.000, C 0.000 }
gfCNCPoint1[15597] = {X 533.9642, Y 4.1116, Z -1.3333, A 0.000, B 0.000, C 0.000 }
gfCNCPoint1[15598] = {X 533.9641, Y 8.1916, Z -1.3333, A 0.000, B 0.000, C 0.000 }
gfCNCPoint1[15599] = {X 543.7544, Y 8.1919, Z -1.3333, A 0.000, B 0.000, C 0.000 }
gfCNCPoint1[15600] = {X 544.6625, Y 8.2703, Z -1.3333, A 0.000, B 0.000, C 0.000 }
gfCNCPoint1[15601] = {X 545.5295, Y 8.5519, Z -1.3333, A 0.000, B 0.000, C 0.000 }
gfCNCPoint1[15602] = {X 546.3102, Y 9.0224, Z -1.3333, A 0.000, B 0.000, C 0.000 }
gfCNCPoint1[15603] = {X 546.9644, Y 9.6572, Z -1.3333, A 0.000, B 0.000, C 0.000 }
gfCNCPoint1[15604] = {X 547.4581, Y 10.4234, Z -1.3333, A 0.000, B 0.000, C 0.000 }
gfCNCPoint1[15605] = {X 547.7658, Y 11.2815, Z -1.3333, A 0.000, B 0.000, C 0.000 }
gfCNCPoint1[15606] = {X 547.8714, Y 12.1869, Z -1.3333, A 0.000, B 0.000, C 0.000 }
gfCNCPoint1[15607] = {X 547.8712, Y 13.0192, Z -1.3333, A 0.000, B 0.000, C 0.000 }
gfCNCPoint1[15608] = {X 547.7727, Y 13.8614, Z -1.3333, A 0.000, B 0.000, C 0.000 }
gfCNCPoint1[15609] = {X 547.4988, Y 14.6639, Z -1.3333, A 0.000, B 0.000, C 0.000 }
gfCNCPoint1[15610] = {X 547.0619, Y 15.3907, Z -1.3333, A 0.000, B 0.000, C 0.000 }
gfCNCPoint1[15611] = {X 546.4816, Y 16.0090, Z -1.3333, A 0.000, B 0.000, C 0.000 }
gfCNCPoint1[15612] = {X 546.4143, Y 16.0657, Z -1.3333, A 0.000, B 0.000, C 0.000 }
gfCNCPoint1[15613] = {X 546.3458, Y 16.1209, Z -1.3333, A 0.000, B 0.000, C 0.000 }
gfCNCPoint1[15614] = {X 546.3426, Y 16.3121, Z -1.3333, A 0.000, B 0.000, C 0.000 }
gfCNCPoint1[15615] = {X 546.3428, Y 41.0663, Z -1.3333, A 0.000, B 0.000, C 0.000 }
gfCNCPoint1[15616] = {X 546.4818, Y 41.1780, Z -1.3333, A 0.000, B 0.000, C 0.000 }
gfCNCPoint1[15617] = {X 547.0682, Y 41.8045, Z -1.3333, A 0.000, B 0.000, C 0.000 }
gfCNCPoint1[15618] = {X 547.5075, Y 42.5417, Z -1.3333, A 0.000, B 0.000, C 0.000 }
gfCNCPoint1[15619] = {X 547.7794, Y 43.3557, Z -1.3333, A 0.000, B 0.000, C 0.000 }
gfCNCPoint1[15620] = {X 547.8714, Y 44.2089, Z -1.3333, A 0.000, B 0.000, C 0.000 }
gfCNCPoint1[15621] = {X 547.8714, Y 44.9999, Z -1.3333, A 0.000, B 0.000, C 0.000 }
gfCNCPoint1[15622] = {X 547.7658, Y 45.9053, Z -1.3333, A 0.000, B 0.000, C 0.000 }
gfCNCPoint1[15623] = {X 547.4581, Y 46.7633, Z -1.3333, A 0.000, B 0.000, C 0.000 }
gfCNCPoint1[15624] = {X 546.9644, Y 47.5296, Z -1.3333, A 0.000, B 0.000, C 0.000 }
gfCNCPoint1[15625] = {X 546.3102, Y 48.1643, Z -1.3333, A 0.000, B 0.000, C 0.000 }
gfCNCPoint1[15626] = {X 545.5294, Y 48.6347, Z -1.3333, A 0.000, B 0.000, C 0.000 }
gfCNCPoint1[15627] = {X 544.6625, Y 48.9163, Z -1.3333, A 0.000, B 0.000, C 0.000 }
gfCNCPoint1[15628] = {X 543.7544, Y 48.9946, Z -1.3333, A 0.000, B 0.000, C 0.000 }
gfCNCPoint1[15629] = {X 523.8755, Y 48.9952, Z -1.3333, A 0.000, B 0.000, C 0.000 }
gfCNCPoint1[15630] = {X 523.3692, Y 49.6263, Z -1.3333, A 0.000, B 0.000, C 0.000 }
gfCNCPoint1[15631] = {X 522.7503, Y 50.1474, Z -1.3333, A 0.000, B 0.000, C 0.000 }
gfCNCPoint1[15632] = {X 522.0422, Y 50.5389, Z -1.3333, A 0.000, B 0.000, C 0.000 }
gfCNCPoint1[15633] = {X 521.2718, Y 50.7859, Z -1.3333, A 0.000, B 0.000, C 0.000 }
gfCNCPoint1[15634] = {X 520.4681, Y 50.8791, Z -1.3333, A 0.000, B 0.000, C 0.000 }
gfCNCPoint1[15635] = {X 519.7998, Y 50.8791, Z -1.3333, A 0.000, B 0.000, C 0.000 }
gfCNCPoint1[15636] = {X 518.9097, Y 50.7788, Z -1.3333, A 0.000, B 0.000, C 0.000 }
gfCNCPoint1[15637] = {X 518.0642, Y 50.4830, Z -1.3333, A 0.000, B 0.000, C 0.000 }
gfCNCPoint1[15638] = {X 517.3058, Y 50.0064, Z -1.3333, A 0.000, B 0.000, C 0.000 }
gfCNCPoint1[15639] = {X 516.6724, Y 49.3731, Z -1.3333, A 0.000, B 0.000, C 0.000 }
gfCNCPoint1[15640] = {X 516.1959, Y 48.6147, Z -1.3333, A 0.000, B 0.000, C 0.000 }
gfCNCPoint1[15641] = {X 515.9001, Y 47.7692, Z -1.3333, A 0.000, B 0.000, C 0.000 }
gfCNCPoint1[15642] = {X 515.7998, Y 46.8791, Z -1.3333, A 0.000, B 0.000, C 0.000 }
gfCNCPoint1[15643] = {X 515.7998, Y 39.9011, Z -1.3333, A 0.000, B 0.000, C 0.000 }
gfCNCPoint1[15644] = {X 515.9001, Y 39.0110, Z -1.3333, A 0.000, B 0.000, C 0.000 }
gfCNCPoint1[15645] = {X 516.1959, Y 38.1655, Z -1.3333, A 0.000, B 0.000, C 0.000 }
gfCNCPoint1[15646] = {X 516.6725, Y 37.4071, Z -1.3333, A 0.000, B 0.000, C 0.000 }
gfCNCPoint1[15647] = {X 517.3059, Y 36.7737, Z -1.3333, A 0.000, B 0.000, C 0.000 }
